       #MyDInt	:= 0;
       #MyWordsinDint[0]	:= "EPICSToPLC"."Word"[#EPICSToPLCDataBlockOffset + 17];
       #MyWordsinDint[1]	:= "EPICSToPLC"."Word"[#EPICSToPLCDataBlockOffset + 18];
       #"P_BlockIcon_LockID" := #MyDInt;    //EPICSName: P_BlockIcon_LockID
    Else
       #DEVICE_PARAM_OK := FALSE; //Invalid Hash
    END_IF;
END_FUNCTION_BLOCK
FUNCTION_BLOCK "DEVTYPE_ICS_HV"
{ S7_Optimized_Access := 'TRUE' }
VERSION : 1.0
   VAR_INPUT
      "OpMode_FreeRun" { ExternalAccessible := 'True'; ExternalVisible := 'False'; ExternalWritable := 'False'; } : BOOL;   //EPICS Status variable: OpMode_FreeRun
      "OpMode_Forced" { ExternalAccessible := 'True'; ExternalVisible := 'False'; ExternalWritable := 'False'; } : BOOL;   //EPICS Status variable: OpMode_Forced
      "Opened" { ExternalAccessible := 'True'; ExternalVisible := 'False'; ExternalWritable := 'False'; } : BOOL;   //EPICS Status variable: Opened
      "Closed" { ExternalAccessible := 'True'; ExternalVisible := 'False'; ExternalWritable := 'False'; } : BOOL;   //EPICS Status variable: Closed
      "ValveColor" { ExternalAccessible := 'True'; ExternalVisible := 'False'; ExternalWritable := 'False'; } : INT;   //EPICS Status variable: ValveColor
      "Inhibit_Manual" { ExternalAccessible := 'True'; ExternalVisible := 'False'; ExternalWritable := 'False'; } : BOOL;   //EPICS Status variable: Inhibit_Manual
      "Inhibit_Force" { ExternalAccessible := 'True'; ExternalVisible := 'False'; ExternalWritable := 'False'; } : BOOL;   //EPICS Status variable: Inhibit_Force
      "Inhibit_Lock" { ExternalAccessible := 'True'; ExternalVisible := 'False'; ExternalWritable := 'False'; } : BOOL;   //EPICS Status variable: Inhibit_Lock
      "EnableFreeRunBtn" { ExternalAccessible := 'True'; ExternalVisible := 'False'; ExternalWritable := 'False'; } : BOOL;   //EPICS Status variable: EnableFreeRunBtn
      "EnableManualBtn" { ExternalAccessible := 'True'; ExternalVisible := 'False'; ExternalWritable := 'False'; } : BOOL;   //EPICS Status variable: EnableManualBtn
      "EnableForcedBtn" { ExternalAccessible := 'True'; ExternalVisible := 'False'; ExternalWritable := 'False'; } : BOOL;   //EPICS Status variable: EnableForcedBtn
      "DevLocked" { ExternalAccessible := 'True'; ExternalVisible := 'False'; ExternalWritable := 'False'; } : BOOL;   //EPICS Status variable: DevLocked
      "Faceplate_LockID" { ExternalAccessible := 'True'; ExternalVisible := 'False'; ExternalWritable := 'False'; } : DINT;   //EPICS Status variable: Faceplate_LockID
      "BlockIcon_LockID" { ExternalAccessible := 'True'; ExternalVisible := 'False'; ExternalWritable := 'False'; } : DINT;   //EPICS Status variable: BlockIcon_LockID
      "LatchAlarm" { ExternalAccessible := 'True'; ExternalVisible := 'False'; ExternalWritable := 'False'; } : BOOL;   //EPICS Status variable: LatchAlarm
      "GroupAlarm" { ExternalAccessible := 'True'; ExternalVisible := 'False'; ExternalWritable := 'False'; } : BOOL;   //EPICS Status variable: GroupAlarm
      "IO_Error" { ExternalAccessible := 'True'; ExternalVisible := 'False'; ExternalWritable := 'False'; } : BOOL;   //EPICS Status variable: IO_Error
      "Input_Module_Error" { ExternalAccessible := 'True'; ExternalVisible := 'False'; ExternalWritable := 'False'; } : BOOL;   //EPICS Status variable: Input_Module_Error
   EPICSToPLCLength { ExternalAccessible := 'False'; ExternalVisible := 'False'; ExternalWritable := 'False'; } : Int;   // Length of device command register array (in words)
   EPICSToPLCDataBlockOffset { ExternalAccessible := 'False'; ExternalVisible := 'False'; ExternalWritable := 'False'; } : Int;   // Offset in EPICS->PLC comms block where this device data resides (in words)
   PLCToEPICSLength { ExternalAccessible := 'False'; ExternalVisible := 'False'; ExternalWritable := 'False'; } : Int;   // Length of device status register array (in words)
   PLCToEPICSDataBlockOffset { ExternalAccessible := 'False'; ExternalVisible := 'False'; ExternalWritable := 'False'; } : Int;   // Offset in PLC->EPICS comms block where this device data resides (in words)
   END_VAR
   VAR_OUTPUT
      "Cmd_FreeRun" { ExternalAccessible := 'True'; ExternalVisible := 'False'; ExternalWritable := 'False'; } : BOOL;   //EPICS Command variable: Cmd_FreeRun
      "Cmd_Force" { ExternalAccessible := 'True'; ExternalVisible := 'False'; ExternalWritable := 'False'; } : BOOL;   //EPICS Command variable: Cmd_Force
      "Cmd_ForceVal" { ExternalAccessible := 'True'; ExternalVisible := 'False'; ExternalWritable := 'False'; } : BOOL;   //EPICS Command variable: Cmd_ForceVal
      "Cmd_AckAlarm" { ExternalAccessible := 'True'; ExternalVisible := 'False'; ExternalWritable := 'False'; } : BOOL;   //EPICS Command variable: Cmd_AckAlarm
      "Cmd_ForceUnlock" { ExternalAccessible := 'True'; ExternalVisible := 'False'; ExternalWritable := 'False'; } : BOOL;   //EPICS Command variable: Cmd_ForceUnlock
      "Cmd_DevLock" { ExternalAccessible := 'True'; ExternalVisible := 'False'; ExternalWritable := 'False'; } : BOOL;   //EPICS Command variable: Cmd_DevLock
      "Cmd_DevUnlock" { ExternalAccessible := 'True'; ExternalVisible := 'False'; ExternalWritable := 'False'; } : BOOL;   //EPICS Command variable: Cmd_DevUnlock
      "P_Faceplate_LockID" { ExternalAccessible := 'True'; ExternalVisible := 'False'; ExternalWritable := 'False'; } : DINT;   //EPICS Parameter variable: P_Faceplate_LockID
      "P_BlockIcon_LockID" { ExternalAccessible := 'True'; ExternalVisible := 'False'; ExternalWritable := 'False'; } : DINT;   //EPICS Parameter variable: P_BlockIcon_LockID
      DEVICE_PARAM_OK { ExternalAccessible := 'False'; ExternalVisible := 'False'; ExternalWritable := 'False'; } : Bool;
   END_VAR
   VAR_IN_OUT
   END_VAR
   Var DB_SPECIFIC
      MyWord { ExternalAccessible := 'False'; ExternalVisible := 'False'; ExternalWritable := 'False'; } : Word;
      MyBytesinWord { ExternalAccessible := 'False'; ExternalVisible := 'False'; ExternalWritable := 'False'; } AT MyWord : Array[0..1] of Byte;
      MyBoolsinWord { ExternalAccessible := 'False'; ExternalVisible := 'False'; ExternalWritable := 'False'; } AT MyWord : Array[0..15] of Bool;
      MyDInt { ExternalAccessible := 'False'; ExternalVisible := 'False'; ExternalWritable := 'False'; } : DInt;
      MyWordsinDint { ExternalAccessible := 'False'; ExternalVisible := 'False'; ExternalWritable := 'False'; } AT MyDInt : Array[0..1] of Word;
      MyReal { ExternalAccessible := 'False'; ExternalVisible := 'False'; ExternalWritable := 'False'; } : Real;
      MyWordsinReal { ExternalAccessible := 'False'; ExternalVisible := 'False'; ExternalWritable := 'False'; } AT MyReal : Array[0..1] of Word;
      MyInt { ExternalAccessible := 'False'; ExternalVisible := 'False'; ExternalWritable := 'False'; } : Int;
      MyWordinInt { ExternalAccessible := 'False'; ExternalVisible := 'False'; ExternalWritable := 'False'; } AT MyInt : Word;
      MyDWord { ExternalAccessible := 'False'; ExternalVisible := 'False'; ExternalWritable := 'False'; } : DWord;
      MyWordsinDWord { ExternalAccessible := 'False'; ExternalVisible := 'False'; ExternalWritable := 'False'; } AT MyDWord : Array[0..1] of Word;
      MyTime { ExternalAccessible := 'False'; ExternalVisible := 'False'; ExternalWritable := 'False'; } : Time;
      MyWordsinTime { ExternalAccessible := 'False'; ExternalVisible := 'False'; ExternalWritable := 'False'; } AT MyTime : Array[0..1] of Word;
      MyString { ExternalAccessible := 'False'; ExternalVisible := 'False'; ExternalWritable := 'False'; } : String[40];
      MyWordsinString { ExternalAccessible := 'False'; ExternalVisible := 'False'; ExternalWritable := 'False'; } AT MyString : Array[0..20] of Word;
   END_VAR
   VAR_TEMP
      HashModbus : DInt;
      HashIFA : DInt;
      HashTIAMap : DInt;
      i : Int;
   END_VAR
    //Author: Miklos Boros (miklos.boros@esss.se), Copyrigth 2017-2020 by European Spallation Source, Lund
    //This block was generated by PLCFactory, please don't change it MANUALLY!
    //Input File Name: Spk-000CDL_Cryo-PLC-010-template-IFA-20220922093722.ifa
    //Generated: 20220922093722
    //According to HASH: 457744924
    //Device type: ICS_HV
    //Description: This function does the variable mapping for a device. All device-variable will be linked to an interface variable defined in this block.

    //********************************************
    //****************HASH check******************
    //********************************************


    #MyWordsinDint[0] := "EPICSToPLC"."Word"[0];
    #MyWordsinDint[1] := "EPICSToPLC"."Word"[1];
    #HashModbus := #MyDInt; //Hash from EPICS/ModbusTCP

    #HashIFA := 457744924; //Hash from Interface Factory as a constant

    #MyWordsinDint[0] := "PLCToEPICS"."Word"[0];
    #MyWordsinDint[1] := "PLCToEPICS"."Word"[1];
    #HashTIAMap := #MyDInt; //Hash from PLCFactory TIA Map


    IF ((#HashIFA = #HashModbus) AND (#HashModbus = #HashTIAMap)) THEN //Check CRCs
        #DEVICE_PARAM_OK := TRUE;
       //##################################### ICS HWI ###############################################
       //############################  ICS Instrument Library     ####################################
       //#  PLC Sample Code in VersionDog: ICS_LIBRARY_MASTER_PLC                                   ##
       //#  CCDB device types: ICS_xxxxx                                                            ##
       //#  EPICS HMI (Block Icons/Faceplates)@ GitLab. Projekt: Cryo / CryogenicsLibrary / CryoLib ##
       //#                                                                                          ##
       //#                          HV - Hand valve with position feedback
       //#                                                                                          ##
       //#                                                                                          ##
       //###########################         Version: 1.3             ################################
       //Author:  Miklos Boros
       //Date:    27-05-2019
       //Version: v1.3
       //Changes:
       //1. Variable Name Unification
       //###########################         Version: 1.0, 1.1, 1.2             ######################
       //Author:  Miklos Boros
       //Date:    28-02-2019
       //Version: v1.2
       //Changes:
       //1. Major review,
       //2. Indent,  unit standardization
       //###########################
       //STATUS BLOCK
       //###########################
       //Operation modes
       //OPI buttons
       //Locking mechanism

    //********************************************
    //*************STATUS VARIABLES***************
    //********************************************


       #MyWord := W#0;
       #MyBoolsinWord[8] := #"OpMode_FreeRun";    //EPICSName: OpMode_FreeRun
       #MyBoolsinWord[9] := #"OpMode_Forced";    //EPICSName: OpMode_Forced
       #MyBoolsinWord[10] := #"Opened";    //EPICSName: Opened
       #MyBoolsinWord[11] := #"Closed";    //EPICSName: Closed
       "PLCToEPICS"."Word"[#PLCToEPICSDataBlockOffset + 0] := #MyWord;

       #MyInt := #"ValveColor";    //EPICSName: ValveColor
       "PLCToEPICS"."Word"[#PLCToEPICSDataBlockOffset + 1] := #MyWordinInt;

       #MyWord := W#0;
       #MyBoolsinWord[8] := #"Inhibit_Manual";    //EPICSName: Inhibit_Manual
       #MyBoolsinWord[9] := #"Inhibit_Force";    //EPICSName: Inhibit_Force
       #MyBoolsinWord[10] := #"Inhibit_Lock";    //EPICSName: Inhibit_Lock
       #MyBoolsinWord[11] := #"EnableFreeRunBtn";    //EPICSName: EnableFreeRunBtn
       #MyBoolsinWord[12] := #"EnableManualBtn";    //EPICSName: EnableManualBtn
       #MyBoolsinWord[13] := #"EnableForcedBtn";    //EPICSName: EnableForcedBtn
       #MyBoolsinWord[14] := #"DevLocked";    //EPICSName: DevLocked
       "PLCToEPICS"."Word"[#PLCToEPICSDataBlockOffset + 2] := #MyWord;

       #MyDInt := #"Faceplate_LockID";    //EPICSName: Faceplate_LockID
       "PLCToEPICS"."Word"[#PLCToEPICSDataBlockOffset + 3] := #MyWordsinDint[0];
       "PLCToEPICS"."Word"[#PLCToEPICSDataBlockOffset + 4] := #MyWordsinDint[1];

       #MyDInt := #"BlockIcon_LockID";    //EPICSName: BlockIcon_LockID
       "PLCToEPICS"."Word"[#PLCToEPICSDataBlockOffset + 5] := #MyWordsinDint[0];
       "PLCToEPICS"."Word"[#PLCToEPICSDataBlockOffset + 6] := #MyWordsinDint[1];

       #MyWord := W#0;
       #MyBoolsinWord[8] := #"LatchAlarm";    //EPICSName: LatchAlarm
       #MyBoolsinWord[9] := #"GroupAlarm";    //EPICSName: GroupAlarm
       #MyBoolsinWord[10] := #"IO_Error";    //EPICSName: IO_Error
       #MyBoolsinWord[11] := #"Input_Module_Error";    //EPICSName: Input_Module_Error
       "PLCToEPICS"."Word"[#PLCToEPICSDataBlockOffset + 7] := #MyWord;

    //********************************************
    //*************COMMAND VARIABLES**************
    //********************************************


       #MyWord := "EPICSToPLC"."Word"[#EPICSToPLCDataBlockOffset + 0];
       "EPICSToPLC"."Word"[#EPICSToPLCDataBlockOffset + 0] := 0;
       #"Cmd_FreeRun" := #MyBoolsinWord[8];    //EPICSName: Cmd_FreeRun
       #"Cmd_Force" := #MyBoolsinWord[9];    //EPICSName: Cmd_Force
       #"Cmd_ForceVal" := #MyBoolsinWord[10];    //EPICSName: Cmd_ForceVal
       #"Cmd_AckAlarm" := #MyBoolsinWord[11];    //EPICSName: Cmd_AckAlarm
       #"Cmd_ForceUnlock" := #MyBoolsinWord[12];    //EPICSName: Cmd_ForceUnlock
       #"Cmd_DevLock" := #MyBoolsinWord[13];    //EPICSName: Cmd_DevLock
       #"Cmd_DevUnlock" := #MyBoolsinWord[14];    //EPICSName: Cmd_DevUnlock

    //********************************************
    //************PARAMETER VARIABLES*************
    //********************************************


       #MyDInt	:= 0;
       #MyWordsinDint[0]	:= "EPICSToPLC"."Word"[#EPICSToPLCDataBlockOffset + 1];
       #MyWordsinDint[1]	:= "EPICSToPLC"."Word"[#EPICSToPLCDataBlockOffset + 2];
       #"P_Faceplate_LockID" := #MyDInt;    //EPICSName: P_Faceplate_LockID

       #MyDInt	:= 0;
       #MyWordsinDint[0]	:= "EPICSToPLC"."Word"[#EPICSToPLCDataBlockOffset + 3];
       #MyWordsinDint[1]	:= "EPICSToPLC"."Word"[#EPICSToPLCDataBlockOffset + 4];
       #"P_BlockIcon_LockID" := #MyDInt;    //EPICSName: P_BlockIcon_LockID
    Else
       #DEVICE_PARAM_OK := FALSE; //Invalid Hash
    END_IF;
END_FUNCTION_BLOCK
FUNCTION_BLOCK "DEVTYPE_ICS_LAKESHORE_TT"
{ S7_Optimized_Access := 'TRUE' }
VERSION : 1.0
   VAR_INPUT
      "OpMode_FreeRun" { ExternalAccessible := 'True'; ExternalVisible := 'False'; ExternalWritable := 'False'; } : BOOL;   //EPICS Status variable: OpMode_FreeRun
      "OpMode_Forced" { ExternalAccessible := 'True'; ExternalVisible := 'False'; ExternalWritable := 'False'; } : BOOL;   //EPICS Status variable: OpMode_Forced
      "Inhibit_Manual" { ExternalAccessible := 'True'; ExternalVisible := 'False'; ExternalWritable := 'False'; } : BOOL;   //EPICS Status variable: Inhibit_Manual
      "Inhibit_Force" { ExternalAccessible := 'True'; ExternalVisible := 'False'; ExternalWritable := 'False'; } : BOOL;   //EPICS Status variable: Inhibit_Force
      "Inhibit_Lock" { ExternalAccessible := 'True'; ExternalVisible := 'False'; ExternalWritable := 'False'; } : BOOL;   //EPICS Status variable: Inhibit_Lock
      "TransmitterColor" { ExternalAccessible := 'True'; ExternalVisible := 'False'; ExternalWritable := 'False'; } : INT;   //EPICS Status variable: TransmitterColor
      "MinTemp" { ExternalAccessible := 'True'; ExternalVisible := 'False'; ExternalWritable := 'False'; } : REAL;   //EPICS Status variable: MinTemp
      "MaxTemp" { ExternalAccessible := 'True'; ExternalVisible := 'False'; ExternalWritable := 'False'; } : REAL;   //EPICS Status variable: MaxTemp
      "EnableFreeRunBtn" { ExternalAccessible := 'True'; ExternalVisible := 'False'; ExternalWritable := 'False'; } : BOOL;   //EPICS Status variable: EnableFreeRunBtn
      "EnableForcedBtn" { ExternalAccessible := 'True'; ExternalVisible := 'False'; ExternalWritable := 'False'; } : BOOL;   //EPICS Status variable: EnableForcedBtn
      "EnableManualBtn" { ExternalAccessible := 'True'; ExternalVisible := 'False'; ExternalWritable := 'False'; } : BOOL;   //EPICS Status variable: EnableManualBtn
      "MeasValue" { ExternalAccessible := 'True'; ExternalVisible := 'False'; ExternalWritable := 'False'; } : REAL;   //EPICS Status variable: MeasValue
      "DevLocked" { ExternalAccessible := 'True'; ExternalVisible := 'False'; ExternalWritable := 'False'; } : BOOL;   //EPICS Status variable: DevLocked
      "Faceplate_LockID" { ExternalAccessible := 'True'; ExternalVisible := 'False'; ExternalWritable := 'False'; } : DINT;   //EPICS Status variable: Faceplate_LockID
      "BlockIcon_LockID" { ExternalAccessible := 'True'; ExternalVisible := 'False'; ExternalWritable := 'False'; } : DINT;   //EPICS Status variable: BlockIcon_LockID
      "LatchAlarm" { ExternalAccessible := 'True'; ExternalVisible := 'False'; ExternalWritable := 'False'; } : BOOL;   //EPICS Status variable: LatchAlarm
      "GroupAlarm" { ExternalAccessible := 'True'; ExternalVisible := 'False'; ExternalWritable := 'False'; } : BOOL;   //EPICS Status variable: GroupAlarm
      "Underrange" { ExternalAccessible := 'True'; ExternalVisible := 'False'; ExternalWritable := 'False'; } : BOOL;   //EPICS Status variable: Underrange
      "Overrange" { ExternalAccessible := 'True'; ExternalVisible := 'False'; ExternalWritable := 'False'; } : BOOL;   //EPICS Status variable: Overrange
      "HIHI" { ExternalAccessible := 'True'; ExternalVisible := 'False'; ExternalWritable := 'False'; } : BOOL;   //EPICS Status variable: HIHI
      "HI" { ExternalAccessible := 'True'; ExternalVisible := 'False'; ExternalWritable := 'False'; } : BOOL;   //EPICS Status variable: HI
      "LO" { ExternalAccessible := 'True'; ExternalVisible := 'False'; ExternalWritable := 'False'; } : BOOL;   //EPICS Status variable: LO
      "LOLO" { ExternalAccessible := 'True'; ExternalVisible := 'False'; ExternalWritable := 'False'; } : BOOL;   //EPICS Status variable: LOLO
      "Param_Error" { ExternalAccessible := 'True'; ExternalVisible := 'False'; ExternalWritable := 'False'; } : BOOL;   //EPICS Status variable: Param_Error
      "PN_Module_Error" { ExternalAccessible := 'True'; ExternalVisible := 'False'; ExternalWritable := 'False'; } : BOOL;   //EPICS Status variable: PN_Module_Error
      "FB_ForceValue" { ExternalAccessible := 'True'; ExternalVisible := 'False'; ExternalWritable := 'False'; } : REAL;   //EPICS Status variable: FB_ForceValue
      "FB_Limit_HIHI" { ExternalAccessible := 'True'; ExternalVisible := 'False'; ExternalWritable := 'False'; } : REAL;   //EPICS Status variable: FB_Limit_HIHI
      "FB_Limit_HI" { ExternalAccessible := 'True'; ExternalVisible := 'False'; ExternalWritable := 'False'; } : REAL;   //EPICS Status variable: FB_Limit_HI
      "FB_Limit_LO" { ExternalAccessible := 'True'; ExternalVisible := 'False'; ExternalWritable := 'False'; } : REAL;   //EPICS Status variable: FB_Limit_LO
      "FB_Limit_LOLO" { ExternalAccessible := 'True'; ExternalVisible := 'False'; ExternalWritable := 'False'; } : REAL;   //EPICS Status variable: FB_Limit_LOLO
   EPICSToPLCLength { ExternalAccessible := 'False'; ExternalVisible := 'False'; ExternalWritable := 'False'; } : Int;   // Length of device command register array (in words)
   EPICSToPLCDataBlockOffset { ExternalAccessible := 'False'; ExternalVisible := 'False'; ExternalWritable := 'False'; } : Int;   // Offset in EPICS->PLC comms block where this device data resides (in words)
   PLCToEPICSLength { ExternalAccessible := 'False'; ExternalVisible := 'False'; ExternalWritable := 'False'; } : Int;   // Length of device status register array (in words)
   PLCToEPICSDataBlockOffset { ExternalAccessible := 'False'; ExternalVisible := 'False'; ExternalWritable := 'False'; } : Int;   // Offset in PLC->EPICS comms block where this device data resides (in words)
   END_VAR
   VAR_OUTPUT
      "Cmd_FreeRun" { ExternalAccessible := 'True'; ExternalVisible := 'False'; ExternalWritable := 'False'; } : BOOL;   //EPICS Command variable: Cmd_FreeRun
      "Cmd_Force" { ExternalAccessible := 'True'; ExternalVisible := 'False'; ExternalWritable := 'False'; } : BOOL;   //EPICS Command variable: Cmd_Force
      "Cmd_ForceVal" { ExternalAccessible := 'True'; ExternalVisible := 'False'; ExternalWritable := 'False'; } : BOOL;   //EPICS Command variable: Cmd_ForceVal
      "Cmd_AckAlarm" { ExternalAccessible := 'True'; ExternalVisible := 'False'; ExternalWritable := 'False'; } : BOOL;   //EPICS Command variable: Cmd_AckAlarm
      "Cmd_ForceUnlock" { ExternalAccessible := 'True'; ExternalVisible := 'False'; ExternalWritable := 'False'; } : BOOL;   //EPICS Command variable: Cmd_ForceUnlock
      "Cmd_DevLock" { ExternalAccessible := 'True'; ExternalVisible := 'False'; ExternalWritable := 'False'; } : BOOL;   //EPICS Command variable: Cmd_DevLock
      "Cmd_DevUnlock" { ExternalAccessible := 'True'; ExternalVisible := 'False'; ExternalWritable := 'False'; } : BOOL;   //EPICS Command variable: Cmd_DevUnlock
      "P_Limit_HIHI" { ExternalAccessible := 'True'; ExternalVisible := 'False'; ExternalWritable := 'False'; } : REAL;   //EPICS Parameter variable: P_Limit_HIHI
      "P_Limit_HI" { ExternalAccessible := 'True'; ExternalVisible := 'False'; ExternalWritable := 'False'; } : REAL;   //EPICS Parameter variable: P_Limit_HI
      "P_Limit_LO" { ExternalAccessible := 'True'; ExternalVisible := 'False'; ExternalWritable := 'False'; } : REAL;   //EPICS Parameter variable: P_Limit_LO
      "P_Limit_LOLO" { ExternalAccessible := 'True'; ExternalVisible := 'False'; ExternalWritable := 'False'; } : REAL;   //EPICS Parameter variable: P_Limit_LOLO
      "P_ForceValue" { ExternalAccessible := 'True'; ExternalVisible := 'False'; ExternalWritable := 'False'; } : REAL;   //EPICS Parameter variable: P_ForceValue
      "P_Faceplate_LockID" { ExternalAccessible := 'True'; ExternalVisible := 'False'; ExternalWritable := 'False'; } : DINT;   //EPICS Parameter variable: P_Faceplate_LockID
      "P_BlockIcon_LockID" { ExternalAccessible := 'True'; ExternalVisible := 'False'; ExternalWritable := 'False'; } : DINT;   //EPICS Parameter variable: P_BlockIcon_LockID
      DEVICE_PARAM_OK { ExternalAccessible := 'False'; ExternalVisible := 'False'; ExternalWritable := 'False'; } : Bool;
   END_VAR
   VAR_IN_OUT
   END_VAR
   Var DB_SPECIFIC
      MyWord { ExternalAccessible := 'False'; ExternalVisible := 'False'; ExternalWritable := 'False'; } : Word;
      MyBytesinWord { ExternalAccessible := 'False'; ExternalVisible := 'False'; ExternalWritable := 'False'; } AT MyWord : Array[0..1] of Byte;
      MyBoolsinWord { ExternalAccessible := 'False'; ExternalVisible := 'False'; ExternalWritable := 'False'; } AT MyWord : Array[0..15] of Bool;
      MyDInt { ExternalAccessible := 'False'; ExternalVisible := 'False'; ExternalWritable := 'False'; } : DInt;
      MyWordsinDint { ExternalAccessible := 'False'; ExternalVisible := 'False'; ExternalWritable := 'False'; } AT MyDInt : Array[0..1] of Word;
      MyReal { ExternalAccessible := 'False'; ExternalVisible := 'False'; ExternalWritable := 'False'; } : Real;
      MyWordsinReal { ExternalAccessible := 'False'; ExternalVisible := 'False'; ExternalWritable := 'False'; } AT MyReal : Array[0..1] of Word;
      MyInt { ExternalAccessible := 'False'; ExternalVisible := 'False'; ExternalWritable := 'False'; } : Int;
      MyWordinInt { ExternalAccessible := 'False'; ExternalVisible := 'False'; ExternalWritable := 'False'; } AT MyInt : Word;
      MyDWord { ExternalAccessible := 'False'; ExternalVisible := 'False'; ExternalWritable := 'False'; } : DWord;
      MyWordsinDWord { ExternalAccessible := 'False'; ExternalVisible := 'False'; ExternalWritable := 'False'; } AT MyDWord : Array[0..1] of Word;
      MyTime { ExternalAccessible := 'False'; ExternalVisible := 'False'; ExternalWritable := 'False'; } : Time;
      MyWordsinTime { ExternalAccessible := 'False'; ExternalVisible := 'False'; ExternalWritable := 'False'; } AT MyTime : Array[0..1] of Word;
      MyString { ExternalAccessible := 'False'; ExternalVisible := 'False'; ExternalWritable := 'False'; } : String[40];
      MyWordsinString { ExternalAccessible := 'False'; ExternalVisible := 'False'; ExternalWritable := 'False'; } AT MyString : Array[0..20] of Word;
   END_VAR
   VAR_TEMP
      HashModbus : DInt;
      HashIFA : DInt;
      HashTIAMap : DInt;
      i : Int;
   END_VAR
    //Author: Miklos Boros (miklos.boros@esss.se), Copyrigth 2017-2020 by European Spallation Source, Lund
    //This block was generated by PLCFactory, please don't change it MANUALLY!
    //Input File Name: Spk-000CDL_Cryo-PLC-010-template-IFA-20220922093722.ifa
    //Generated: 20220922093722
    //According to HASH: 457744924
    //Device type: ICS_LAKESHORE_TT
    //Description: This function does the variable mapping for a device. All device-variable will be linked to an interface variable defined in this block.

    //********************************************
    //****************HASH check******************
    //********************************************


    #MyWordsinDint[0] := "EPICSToPLC"."Word"[0];
    #MyWordsinDint[1] := "EPICSToPLC"."Word"[1];
    #HashModbus := #MyDInt; //Hash from EPICS/ModbusTCP

    #HashIFA := 457744924; //Hash from Interface Factory as a constant

    #MyWordsinDint[0] := "PLCToEPICS"."Word"[0];
    #MyWordsinDint[1] := "PLCToEPICS"."Word"[1];
    #HashTIAMap := #MyDInt; //Hash from PLCFactory TIA Map


    IF ((#HashIFA = #HashModbus) AND (#HashModbus = #HashTIAMap)) THEN //Check CRCs
        #DEVICE_PARAM_OK := TRUE;
       //##################################### ICS HWI ###############################################
       //############################  ICS Instrument Library     ####################################
       //#  PLC Sample Code in VersionDog: ICS_LIBRARY_MASTER_PLC                                   ##
       //#  CCDB device types: ICS_xxxxx                                                            ##
       //#  EPICS HMI (Block Icons/Faceplates)@ GitLab. Projekt: Cryo / CryogenicsLibrary / CryoLib ##
       //#                                                                                          ##
       //#                      TT - Temperature Transmitter in K with Lakeshore                    ##
       //#                                                                                          ##
       //#                                                                                          ##
       //###########################         Version: 1.4             ################################
       //Author:  Miklos Boros
       //Date:    16-12-2019
       //Version: v1.4
       //Changes:
       //1. Modified TT for direct Temp measurement with Lakeshore
       //###########################         Version: 1.3             ################################
       //Author:  Miklos Boros
       //Date:    27-05-2019
       //Version: v1.3
       //Changes:
       //1. Variable Name Unification
       //###########################         Version: 1.2             ################################
       //Author:  Miklos Boros
       //Date:    28-02-2019
       //Version: v1.2
       //Changes:
       //1. Major review,
       //2. Indent,  unit standardization
       //###########################         Version: 1.1             ################################
       //Author:  Miklos Boros, Marino Vojneski
       //Date:    12-06-2018
       //Version: v1.1
       //Changes:
       //1. Modified Alarm Signal section to be compatible with new format.
       //########################### Version: 1.0             ########################################
       //Author:  Miklos Boros
       //Date:    25-01-2018
       //Version: v1.0
       //###########################
       //STATUS BLOCK
       //###########################
       //Operation modes
       //OPI buttons
       //Limits

    //********************************************
    //*************STATUS VARIABLES***************
    //********************************************


       #MyWord := W#0;
       #MyBoolsinWord[8] := #"OpMode_FreeRun";    //EPICSName: OpMode_FreeRun
       #MyBoolsinWord[9] := #"OpMode_Forced";    //EPICSName: OpMode_Forced
       #MyBoolsinWord[10] := #"Inhibit_Manual";    //EPICSName: Inhibit_Manual
       #MyBoolsinWord[11] := #"Inhibit_Force";    //EPICSName: Inhibit_Force
       #MyBoolsinWord[12] := #"Inhibit_Lock";    //EPICSName: Inhibit_Lock
       "PLCToEPICS"."Word"[#PLCToEPICSDataBlockOffset + 0] := #MyWord;

       #MyInt := #"TransmitterColor";    //EPICSName: TransmitterColor
       "PLCToEPICS"."Word"[#PLCToEPICSDataBlockOffset + 1] := #MyWordinInt;

       #MyReal := #"MinTemp";    //EPICSName: MinTemp
       "PLCToEPICS"."Word"[#PLCToEPICSDataBlockOffset + 2] := #MyWordsinReal[0];
       "PLCToEPICS"."Word"[#PLCToEPICSDataBlockOffset + 3] := #MyWordsinReal[1];

       #MyReal := #"MaxTemp";    //EPICSName: MaxTemp
       "PLCToEPICS"."Word"[#PLCToEPICSDataBlockOffset + 4] := #MyWordsinReal[0];
       "PLCToEPICS"."Word"[#PLCToEPICSDataBlockOffset + 5] := #MyWordsinReal[1];

       #MyWord := W#0;
       #MyBoolsinWord[8] := #"EnableFreeRunBtn";    //EPICSName: EnableFreeRunBtn
       #MyBoolsinWord[9] := #"EnableForcedBtn";    //EPICSName: EnableForcedBtn
       #MyBoolsinWord[10] := #"EnableManualBtn";    //EPICSName: EnableManualBtn
       "PLCToEPICS"."Word"[#PLCToEPICSDataBlockOffset + 6] := #MyWord;

       #MyReal := #"MeasValue";    //EPICSName: MeasValue
       "PLCToEPICS"."Word"[#PLCToEPICSDataBlockOffset + 7] := #MyWordsinReal[0];
       "PLCToEPICS"."Word"[#PLCToEPICSDataBlockOffset + 8] := #MyWordsinReal[1];

       #MyWord := W#0;
       #MyBoolsinWord[8] := #"DevLocked";    //EPICSName: DevLocked
       "PLCToEPICS"."Word"[#PLCToEPICSDataBlockOffset + 9] := #MyWord;

       #MyDInt := #"Faceplate_LockID";    //EPICSName: Faceplate_LockID
       "PLCToEPICS"."Word"[#PLCToEPICSDataBlockOffset + 10] := #MyWordsinDint[0];
       "PLCToEPICS"."Word"[#PLCToEPICSDataBlockOffset + 11] := #MyWordsinDint[1];

       #MyDInt := #"BlockIcon_LockID";    //EPICSName: BlockIcon_LockID
       "PLCToEPICS"."Word"[#PLCToEPICSDataBlockOffset + 12] := #MyWordsinDint[0];
       "PLCToEPICS"."Word"[#PLCToEPICSDataBlockOffset + 13] := #MyWordsinDint[1];

       #MyWord := W#0;
       #MyBoolsinWord[8] := #"LatchAlarm";    //EPICSName: LatchAlarm
       #MyBoolsinWord[9] := #"GroupAlarm";    //EPICSName: GroupAlarm
       #MyBoolsinWord[10] := #"Underrange";    //EPICSName: Underrange
       #MyBoolsinWord[11] := #"Overrange";    //EPICSName: Overrange
       #MyBoolsinWord[12] := #"HIHI";    //EPICSName: HIHI
       #MyBoolsinWord[13] := #"HI";    //EPICSName: HI
       #MyBoolsinWord[14] := #"LO";    //EPICSName: LO
       #MyBoolsinWord[15] := #"LOLO";    //EPICSName: LOLO
       #MyBoolsinWord[0] := #"Param_Error";    //EPICSName: Param_Error
       #MyBoolsinWord[1] := #"PN_Module_Error";    //EPICSName: PN_Module_Error
       "PLCToEPICS"."Word"[#PLCToEPICSDataBlockOffset + 14] := #MyWord;

       #MyReal := #"FB_ForceValue";    //EPICSName: FB_ForceValue
       "PLCToEPICS"."Word"[#PLCToEPICSDataBlockOffset + 15] := #MyWordsinReal[0];
       "PLCToEPICS"."Word"[#PLCToEPICSDataBlockOffset + 16] := #MyWordsinReal[1];

       #MyReal := #"FB_Limit_HIHI";    //EPICSName: FB_Limit_HIHI
       "PLCToEPICS"."Word"[#PLCToEPICSDataBlockOffset + 17] := #MyWordsinReal[0];
       "PLCToEPICS"."Word"[#PLCToEPICSDataBlockOffset + 18] := #MyWordsinReal[1];

       #MyReal := #"FB_Limit_HI";    //EPICSName: FB_Limit_HI
       "PLCToEPICS"."Word"[#PLCToEPICSDataBlockOffset + 19] := #MyWordsinReal[0];
       "PLCToEPICS"."Word"[#PLCToEPICSDataBlockOffset + 20] := #MyWordsinReal[1];

       #MyReal := #"FB_Limit_LO";    //EPICSName: FB_Limit_LO
       "PLCToEPICS"."Word"[#PLCToEPICSDataBlockOffset + 21] := #MyWordsinReal[0];
       "PLCToEPICS"."Word"[#PLCToEPICSDataBlockOffset + 22] := #MyWordsinReal[1];

       #MyReal := #"FB_Limit_LOLO";    //EPICSName: FB_Limit_LOLO
       "PLCToEPICS"."Word"[#PLCToEPICSDataBlockOffset + 23] := #MyWordsinReal[0];
       "PLCToEPICS"."Word"[#PLCToEPICSDataBlockOffset + 24] := #MyWordsinReal[1];

    //********************************************
    //*************COMMAND VARIABLES**************
    //********************************************


       #MyWord := "EPICSToPLC"."Word"[#EPICSToPLCDataBlockOffset + 0];
       "EPICSToPLC"."Word"[#EPICSToPLCDataBlockOffset + 0] := 0;
       #"Cmd_FreeRun" := #MyBoolsinWord[8];    //EPICSName: Cmd_FreeRun
       #"Cmd_Force" := #MyBoolsinWord[9];    //EPICSName: Cmd_Force
       #"Cmd_ForceVal" := #MyBoolsinWord[10];    //EPICSName: Cmd_ForceVal
       #"Cmd_AckAlarm" := #MyBoolsinWord[11];    //EPICSName: Cmd_AckAlarm
       #"Cmd_ForceUnlock" := #MyBoolsinWord[12];    //EPICSName: Cmd_ForceUnlock
       #"Cmd_DevLock" := #MyBoolsinWord[13];    //EPICSName: Cmd_DevLock
       #"Cmd_DevUnlock" := #MyBoolsinWord[14];    //EPICSName: Cmd_DevUnlock

    //********************************************
    //************PARAMETER VARIABLES*************
    //********************************************


       #MyReal	:= 0.0;
       #MyWordsinReal[0]	:= "EPICSToPLC"."Word"[#EPICSToPLCDataBlockOffset + 1];
       #MyWordsinReal[1]	:= "EPICSToPLC"."Word"[#EPICSToPLCDataBlockOffset + 2];
       #"P_Limit_HIHI" := #MyReal;    //EPICSName: P_Limit_HIHI

       #MyReal	:= 0.0;
       #MyWordsinReal[0]	:= "EPICSToPLC"."Word"[#EPICSToPLCDataBlockOffset + 3];
       #MyWordsinReal[1]	:= "EPICSToPLC"."Word"[#EPICSToPLCDataBlockOffset + 4];
       #"P_Limit_HI" := #MyReal;    //EPICSName: P_Limit_HI

       #MyReal	:= 0.0;
       #MyWordsinReal[0]	:= "EPICSToPLC"."Word"[#EPICSToPLCDataBlockOffset + 5];
       #MyWordsinReal[1]	:= "EPICSToPLC"."Word"[#EPICSToPLCDataBlockOffset + 6];
       #"P_Limit_LO" := #MyReal;    //EPICSName: P_Limit_LO

       #MyReal	:= 0.0;
       #MyWordsinReal[0]	:= "EPICSToPLC"."Word"[#EPICSToPLCDataBlockOffset + 7];
       #MyWordsinReal[1]	:= "EPICSToPLC"."Word"[#EPICSToPLCDataBlockOffset + 8];
       #"P_Limit_LOLO" := #MyReal;    //EPICSName: P_Limit_LOLO

       #MyReal	:= 0.0;
       #MyWordsinReal[0]	:= "EPICSToPLC"."Word"[#EPICSToPLCDataBlockOffset + 9];
       #MyWordsinReal[1]	:= "EPICSToPLC"."Word"[#EPICSToPLCDataBlockOffset + 10];
       #"P_ForceValue" := #MyReal;    //EPICSName: P_ForceValue

       #MyDInt	:= 0;
       #MyWordsinDint[0]	:= "EPICSToPLC"."Word"[#EPICSToPLCDataBlockOffset + 11];
       #MyWordsinDint[1]	:= "EPICSToPLC"."Word"[#EPICSToPLCDataBlockOffset + 12];
       #"P_Faceplate_LockID" := #MyDInt;    //EPICSName: P_Faceplate_LockID

       #MyDInt	:= 0;
       #MyWordsinDint[0]	:= "EPICSToPLC"."Word"[#EPICSToPLCDataBlockOffset + 13];
       #MyWordsinDint[1]	:= "EPICSToPLC"."Word"[#EPICSToPLCDataBlockOffset + 14];
       #"P_BlockIcon_LockID" := #MyDInt;    //EPICSName: P_BlockIcon_LockID
    Else
       #DEVICE_PARAM_OK := FALSE; //Invalid Hash
    END_IF;
END_FUNCTION_BLOCK
FUNCTION_BLOCK "DEVTYPE_ICS_LT"
{ S7_Optimized_Access := 'TRUE' }
VERSION : 1.0
   VAR_INPUT
      "OpMode_FreeRun" { ExternalAccessible := 'True'; ExternalVisible := 'False'; ExternalWritable := 'False'; } : BOOL;   //EPICS Status variable: OpMode_FreeRun
      "OpMode_Forced" { ExternalAccessible := 'True'; ExternalVisible := 'False'; ExternalWritable := 'False'; } : BOOL;   //EPICS Status variable: OpMode_Forced
      "Inhibit_Manual" { ExternalAccessible := 'True'; ExternalVisible := 'False'; ExternalWritable := 'False'; } : BOOL;   //EPICS Status variable: Inhibit_Manual
      "Inhibit_Force" { ExternalAccessible := 'True'; ExternalVisible := 'False'; ExternalWritable := 'False'; } : BOOL;   //EPICS Status variable: Inhibit_Force
      "Inhibit_Lock" { ExternalAccessible := 'True'; ExternalVisible := 'False'; ExternalWritable := 'False'; } : BOOL;   //EPICS Status variable: Inhibit_Lock
      "TransmitterColor" { ExternalAccessible := 'True'; ExternalVisible := 'False'; ExternalWritable := 'False'; } : INT;   //EPICS Status variable: TransmitterColor
      "EnableFreeRunBtn" { ExternalAccessible := 'True'; ExternalVisible := 'False'; ExternalWritable := 'False'; } : BOOL;   //EPICS Status variable: EnableFreeRunBtn
      "EnableForcedBtn" { ExternalAccessible := 'True'; ExternalVisible := 'False'; ExternalWritable := 'False'; } : BOOL;   //EPICS Status variable: EnableForcedBtn
      "EnableManualBtn" { ExternalAccessible := 'True'; ExternalVisible := 'False'; ExternalWritable := 'False'; } : BOOL;   //EPICS Status variable: EnableManualBtn
      "ScaleLOW" { ExternalAccessible := 'True'; ExternalVisible := 'False'; ExternalWritable := 'False'; } : REAL;   //EPICS Status variable: ScaleLOW
      "ScaleHIGH" { ExternalAccessible := 'True'; ExternalVisible := 'False'; ExternalWritable := 'False'; } : REAL;   //EPICS Status variable: ScaleHIGH
      "MeasValue" { ExternalAccessible := 'True'; ExternalVisible := 'False'; ExternalWritable := 'False'; } : REAL;   //EPICS Status variable: MeasValue
      "RAWValue" { ExternalAccessible := 'True'; ExternalVisible := 'False'; ExternalWritable := 'False'; } : REAL;   //EPICS Status variable: RAWValue
      "DevLocked" { ExternalAccessible := 'True'; ExternalVisible := 'False'; ExternalWritable := 'False'; } : BOOL;   //EPICS Status variable: DevLocked
      "Faceplate_LockID" { ExternalAccessible := 'True'; ExternalVisible := 'False'; ExternalWritable := 'False'; } : DINT;   //EPICS Status variable: Faceplate_LockID
      "BlockIcon_LockID" { ExternalAccessible := 'True'; ExternalVisible := 'False'; ExternalWritable := 'False'; } : DINT;   //EPICS Status variable: BlockIcon_LockID
      "LatchAlarm" { ExternalAccessible := 'True'; ExternalVisible := 'False'; ExternalWritable := 'False'; } : BOOL;   //EPICS Status variable: LatchAlarm
      "GroupAlarm" { ExternalAccessible := 'True'; ExternalVisible := 'False'; ExternalWritable := 'False'; } : BOOL;   //EPICS Status variable: GroupAlarm
      "Underrange" { ExternalAccessible := 'True'; ExternalVisible := 'False'; ExternalWritable := 'False'; } : BOOL;   //EPICS Status variable: Underrange
      "Overrange" { ExternalAccessible := 'True'; ExternalVisible := 'False'; ExternalWritable := 'False'; } : BOOL;   //EPICS Status variable: Overrange
      "HIHI" { ExternalAccessible := 'True'; ExternalVisible := 'False'; ExternalWritable := 'False'; } : BOOL;   //EPICS Status variable: HIHI
      "HI" { ExternalAccessible := 'True'; ExternalVisible := 'False'; ExternalWritable := 'False'; } : BOOL;   //EPICS Status variable: HI
      "LO" { ExternalAccessible := 'True'; ExternalVisible := 'False'; ExternalWritable := 'False'; } : BOOL;   //EPICS Status variable: LO
      "LOLO" { ExternalAccessible := 'True'; ExternalVisible := 'False'; ExternalWritable := 'False'; } : BOOL;   //EPICS Status variable: LOLO
      "IO_Error" { ExternalAccessible := 'True'; ExternalVisible := 'False'; ExternalWritable := 'False'; } : BOOL;   //EPICS Status variable: IO_Error
      "Module_Error" { ExternalAccessible := 'True'; ExternalVisible := 'False'; ExternalWritable := 'False'; } : BOOL;   //EPICS Status variable: Module_Error
      "Param_Error" { ExternalAccessible := 'True'; ExternalVisible := 'False'; ExternalWritable := 'False'; } : BOOL;   //EPICS Status variable: Param_Error
      "FB_ForceValue" { ExternalAccessible := 'True'; ExternalVisible := 'False'; ExternalWritable := 'False'; } : REAL;   //EPICS Status variable: FB_ForceValue
      "FB_Limit_HIHI" { ExternalAccessible := 'True'; ExternalVisible := 'False'; ExternalWritable := 'False'; } : REAL;   //EPICS Status variable: FB_Limit_HIHI
      "FB_Limit_HI" { ExternalAccessible := 'True'; ExternalVisible := 'False'; ExternalWritable := 'False'; } : REAL;   //EPICS Status variable: FB_Limit_HI
      "FB_Limit_LO" { ExternalAccessible := 'True'; ExternalVisible := 'False'; ExternalWritable := 'False'; } : REAL;   //EPICS Status variable: FB_Limit_LO
      "FB_Limit_LOLO" { ExternalAccessible := 'True'; ExternalVisible := 'False'; ExternalWritable := 'False'; } : REAL;   //EPICS Status variable: FB_Limit_LOLO
      "Timer_enabled" { ExternalAccessible := 'True'; ExternalVisible := 'False'; ExternalWritable := 'False'; } : BOOL;   //EPICS Status variable: Timer_enabled
      "T_triggered" { ExternalAccessible := 'True'; ExternalVisible := 'False'; ExternalWritable := 'False'; } : BOOL;   //EPICS Status variable: T_triggered
      "T_running" { ExternalAccessible := 'True'; ExternalVisible := 'False'; ExternalWritable := 'False'; } : INT;   //EPICS Status variable: T_running
      "F_enabled" { ExternalAccessible := 'True'; ExternalVisible := 'False'; ExternalWritable := 'False'; } : BOOL;   //EPICS Status variable: F_enabled
      "FiltedValue" { ExternalAccessible := 'True'; ExternalVisible := 'False'; ExternalWritable := 'False'; } : REAL;   //EPICS Status variable: FiltedValue
   EPICSToPLCLength { ExternalAccessible := 'False'; ExternalVisible := 'False'; ExternalWritable := 'False'; } : Int;   // Length of device command register array (in words)
   EPICSToPLCDataBlockOffset { ExternalAccessible := 'False'; ExternalVisible := 'False'; ExternalWritable := 'False'; } : Int;   // Offset in EPICS->PLC comms block where this device data resides (in words)
   PLCToEPICSLength { ExternalAccessible := 'False'; ExternalVisible := 'False'; ExternalWritable := 'False'; } : Int;   // Length of device status register array (in words)
   PLCToEPICSDataBlockOffset { ExternalAccessible := 'False'; ExternalVisible := 'False'; ExternalWritable := 'False'; } : Int;   // Offset in PLC->EPICS comms block where this device data resides (in words)
   END_VAR
   VAR_OUTPUT
      "Cmd_FreeRun" { ExternalAccessible := 'True'; ExternalVisible := 'False'; ExternalWritable := 'False'; } : BOOL;   //EPICS Command variable: Cmd_FreeRun
      "Cmd_Force" { ExternalAccessible := 'True'; ExternalVisible := 'False'; ExternalWritable := 'False'; } : BOOL;   //EPICS Command variable: Cmd_Force
      "Cmd_ForceVal" { ExternalAccessible := 'True'; ExternalVisible := 'False'; ExternalWritable := 'False'; } : BOOL;   //EPICS Command variable: Cmd_ForceVal
      "Cmd_AckAlarm" { ExternalAccessible := 'True'; ExternalVisible := 'False'; ExternalWritable := 'False'; } : BOOL;   //EPICS Command variable: Cmd_AckAlarm
      "Cmd_ForceUnlock" { ExternalAccessible := 'True'; ExternalVisible := 'False'; ExternalWritable := 'False'; } : BOOL;   //EPICS Command variable: Cmd_ForceUnlock
      "Cmd_DevLock" { ExternalAccessible := 'True'; ExternalVisible := 'False'; ExternalWritable := 'False'; } : BOOL;   //EPICS Command variable: Cmd_DevLock
      "Cmd_DevUnlock" { ExternalAccessible := 'True'; ExternalVisible := 'False'; ExternalWritable := 'False'; } : BOOL;   //EPICS Command variable: Cmd_DevUnlock
      "P_Limit_HIHI" { ExternalAccessible := 'True'; ExternalVisible := 'False'; ExternalWritable := 'False'; } : REAL;   //EPICS Parameter variable: P_Limit_HIHI
      "P_Limit_HI" { ExternalAccessible := 'True'; ExternalVisible := 'False'; ExternalWritable := 'False'; } : REAL;   //EPICS Parameter variable: P_Limit_HI
      "P_Limit_LO" { ExternalAccessible := 'True'; ExternalVisible := 'False'; ExternalWritable := 'False'; } : REAL;   //EPICS Parameter variable: P_Limit_LO
      "P_Limit_LOLO" { ExternalAccessible := 'True'; ExternalVisible := 'False'; ExternalWritable := 'False'; } : REAL;   //EPICS Parameter variable: P_Limit_LOLO
      "P_ForceValue" { ExternalAccessible := 'True'; ExternalVisible := 'False'; ExternalWritable := 'False'; } : REAL;   //EPICS Parameter variable: P_ForceValue
      "P_Faceplate_LockID" { ExternalAccessible := 'True'; ExternalVisible := 'False'; ExternalWritable := 'False'; } : DINT;   //EPICS Parameter variable: P_Faceplate_LockID
      "P_BlockIcon_LockID" { ExternalAccessible := 'True'; ExternalVisible := 'False'; ExternalWritable := 'False'; } : DINT;   //EPICS Parameter variable: P_BlockIcon_LockID
      "T_period" { ExternalAccessible := 'True'; ExternalVisible := 'False'; ExternalWritable := 'False'; } : INT;   //EPICS Parameter variable: T_period
      "F_interval" { ExternalAccessible := 'True'; ExternalVisible := 'False'; ExternalWritable := 'False'; } : INT;   //EPICS Parameter variable: F_interval
      "F_buffer" { ExternalAccessible := 'True'; ExternalVisible := 'False'; ExternalWritable := 'False'; } : INT;   //EPICS Parameter variable: F_buffer
      "F_Enable" { ExternalAccessible := 'True'; ExternalVisible := 'False'; ExternalWritable := 'False'; } : BOOL;   //EPICS Parameter variable: F_Enable
      "P_RampUPSpeed" { ExternalAccessible := 'True'; ExternalVisible := 'False'; ExternalWritable := 'False'; } : REAL;   //EPICS Parameter variable: P_RampUPSpeed
      "P_RampDNSpeed" { ExternalAccessible := 'True'; ExternalVisible := 'False'; ExternalWritable := 'False'; } : REAL;   //EPICS Parameter variable: P_RampDNSpeed
      DEVICE_PARAM_OK { ExternalAccessible := 'False'; ExternalVisible := 'False'; ExternalWritable := 'False'; } : Bool;
   END_VAR
   VAR_IN_OUT
   END_VAR
   Var DB_SPECIFIC
      MyWord { ExternalAccessible := 'False'; ExternalVisible := 'False'; ExternalWritable := 'False'; } : Word;
      MyBytesinWord { ExternalAccessible := 'False'; ExternalVisible := 'False'; ExternalWritable := 'False'; } AT MyWord : Array[0..1] of Byte;
      MyBoolsinWord { ExternalAccessible := 'False'; ExternalVisible := 'False'; ExternalWritable := 'False'; } AT MyWord : Array[0..15] of Bool;
      MyDInt { ExternalAccessible := 'False'; ExternalVisible := 'False'; ExternalWritable := 'False'; } : DInt;
      MyWordsinDint { ExternalAccessible := 'False'; ExternalVisible := 'False'; ExternalWritable := 'False'; } AT MyDInt : Array[0..1] of Word;
      MyReal { ExternalAccessible := 'False'; ExternalVisible := 'False'; ExternalWritable := 'False'; } : Real;
      MyWordsinReal { ExternalAccessible := 'False'; ExternalVisible := 'False'; ExternalWritable := 'False'; } AT MyReal : Array[0..1] of Word;
      MyInt { ExternalAccessible := 'False'; ExternalVisible := 'False'; ExternalWritable := 'False'; } : Int;
      MyWordinInt { ExternalAccessible := 'False'; ExternalVisible := 'False'; ExternalWritable := 'False'; } AT MyInt : Word;
      MyDWord { ExternalAccessible := 'False'; ExternalVisible := 'False'; ExternalWritable := 'False'; } : DWord;
      MyWordsinDWord { ExternalAccessible := 'False'; ExternalVisible := 'False'; ExternalWritable := 'False'; } AT MyDWord : Array[0..1] of Word;
      MyTime { ExternalAccessible := 'False'; ExternalVisible := 'False'; ExternalWritable := 'False'; } : Time;
      MyWordsinTime { ExternalAccessible := 'False'; ExternalVisible := 'False'; ExternalWritable := 'False'; } AT MyTime : Array[0..1] of Word;
      MyString { ExternalAccessible := 'False'; ExternalVisible := 'False'; ExternalWritable := 'False'; } : String[40];
      MyWordsinString { ExternalAccessible := 'False'; ExternalVisible := 'False'; ExternalWritable := 'False'; } AT MyString : Array[0..20] of Word;
   END_VAR
   VAR_TEMP
      HashModbus : DInt;
      HashIFA : DInt;
      HashTIAMap : DInt;
      i : Int;
   END_VAR
    //Author: Miklos Boros (miklos.boros@esss.se), Copyrigth 2017-2020 by European Spallation Source, Lund
    //This block was generated by PLCFactory, please don't change it MANUALLY!
    //Input File Name: Spk-000CDL_Cryo-PLC-010-template-IFA-20220922093722.ifa
    //Generated: 20220922093722
    //According to HASH: 457744924
    //Device type: ICS_LT
    //Description: This function does the variable mapping for a device. All device-variable will be linked to an interface variable defined in this block.

    //********************************************
    //****************HASH check******************
    //********************************************


    #MyWordsinDint[0] := "EPICSToPLC"."Word"[0];
    #MyWordsinDint[1] := "EPICSToPLC"."Word"[1];
    #HashModbus := #MyDInt; //Hash from EPICS/ModbusTCP

    #HashIFA := 457744924; //Hash from Interface Factory as a constant

    #MyWordsinDint[0] := "PLCToEPICS"."Word"[0];
    #MyWordsinDint[1] := "PLCToEPICS"."Word"[1];
    #HashTIAMap := #MyDInt; //Hash from PLCFactory TIA Map


    IF ((#HashIFA = #HashModbus) AND (#HashModbus = #HashTIAMap)) THEN //Check CRCs
        #DEVICE_PARAM_OK := TRUE;
       //##################################### ICS HWI ###############################################
       //############################  ICS Instrument Library     ####################################
       //#  PLC Sample Code in VersionDog: ICS_LIBRARY_MASTER_PLC                                   ##
       //#  CCDB device types: ICS_xxxxx                                                            ##
       //#  EPICS HMI (Block Icons/Faceplates)@ GitLab. Projekt: Cryo / CryogenicsLibrary / CryoLib ##
       //#                                                                                          ##
       //#                          LT- Level Transmitter in percent                                ##
       //#                                                                                          ##
       //#                                                                                          ##
       //###########################         Version: 1.4             ################################
       //Author:  Emilio Asensi
       //Date:    06-09-2022
       //Version: v1.4
       //Changes:
       //1. Added pvs for timer, filter and ramping speed
       //###########################         Version: 1.3             ################################
       //Author:  Miklos Boros
       //Date:    27-05-2019
       //Version: v1.3
       //Changes:
       //1. Variable Name Unification
       //###########################         Version: 1.2             ################################
       //Author:  Miklos Boros
       //Date:    28-02-2019
       //Version: v1.2
       //Changes:
       //1. Major review,
       //2. Indent,  unit standardization
       //###########################         Version: 1.1             ################################
       //Author:  Miklos Boros, Marino Vojneski
       //Date:    12-06-2018
       //Version: v1.1
       //Changes:
       //1. Modified Alarm Signal section to be compatible with new format.
       //########################### Version: 1.0             ########################################
       //Author:  Miklos Boros
       //Date:    25-01-2018
       //Version: v1.0
       //###########################
       //STATUS BLOCK
       //###########################
       //Operation modes
       //OPI buttons
       //Limits

    //********************************************
    //*************STATUS VARIABLES***************
    //********************************************


       #MyWord := W#0;
       #MyBoolsinWord[8] := #"OpMode_FreeRun";    //EPICSName: OpMode_FreeRun
       #MyBoolsinWord[9] := #"OpMode_Forced";    //EPICSName: OpMode_Forced
       #MyBoolsinWord[10] := #"Inhibit_Manual";    //EPICSName: Inhibit_Manual
       #MyBoolsinWord[11] := #"Inhibit_Force";    //EPICSName: Inhibit_Force
       #MyBoolsinWord[12] := #"Inhibit_Lock";    //EPICSName: Inhibit_Lock
       "PLCToEPICS"."Word"[#PLCToEPICSDataBlockOffset + 0] := #MyWord;

       #MyInt := #"TransmitterColor";    //EPICSName: TransmitterColor
       "PLCToEPICS"."Word"[#PLCToEPICSDataBlockOffset + 1] := #MyWordinInt;

       #MyWord := W#0;
       #MyBoolsinWord[8] := #"EnableFreeRunBtn";    //EPICSName: EnableFreeRunBtn
       #MyBoolsinWord[9] := #"EnableForcedBtn";    //EPICSName: EnableForcedBtn
       #MyBoolsinWord[10] := #"EnableManualBtn";    //EPICSName: EnableManualBtn
       "PLCToEPICS"."Word"[#PLCToEPICSDataBlockOffset + 2] := #MyWord;

       #MyReal := #"ScaleLOW";    //EPICSName: ScaleLOW
       "PLCToEPICS"."Word"[#PLCToEPICSDataBlockOffset + 3] := #MyWordsinReal[0];
       "PLCToEPICS"."Word"[#PLCToEPICSDataBlockOffset + 4] := #MyWordsinReal[1];

       #MyReal := #"ScaleHIGH";    //EPICSName: ScaleHIGH
       "PLCToEPICS"."Word"[#PLCToEPICSDataBlockOffset + 5] := #MyWordsinReal[0];
       "PLCToEPICS"."Word"[#PLCToEPICSDataBlockOffset + 6] := #MyWordsinReal[1];

       #MyReal := #"MeasValue";    //EPICSName: MeasValue
       "PLCToEPICS"."Word"[#PLCToEPICSDataBlockOffset + 7] := #MyWordsinReal[0];
       "PLCToEPICS"."Word"[#PLCToEPICSDataBlockOffset + 8] := #MyWordsinReal[1];

       #MyReal := #"RAWValue";    //EPICSName: RAWValue
       "PLCToEPICS"."Word"[#PLCToEPICSDataBlockOffset + 9] := #MyWordsinReal[0];
       "PLCToEPICS"."Word"[#PLCToEPICSDataBlockOffset + 10] := #MyWordsinReal[1];

       #MyWord := W#0;
       #MyBoolsinWord[8] := #"DevLocked";    //EPICSName: DevLocked
       "PLCToEPICS"."Word"[#PLCToEPICSDataBlockOffset + 11] := #MyWord;

       #MyDInt := #"Faceplate_LockID";    //EPICSName: Faceplate_LockID
       "PLCToEPICS"."Word"[#PLCToEPICSDataBlockOffset + 12] := #MyWordsinDint[0];
       "PLCToEPICS"."Word"[#PLCToEPICSDataBlockOffset + 13] := #MyWordsinDint[1];

       #MyDInt := #"BlockIcon_LockID";    //EPICSName: BlockIcon_LockID
       "PLCToEPICS"."Word"[#PLCToEPICSDataBlockOffset + 14] := #MyWordsinDint[0];
       "PLCToEPICS"."Word"[#PLCToEPICSDataBlockOffset + 15] := #MyWordsinDint[1];

       #MyWord := W#0;
       #MyBoolsinWord[8] := #"LatchAlarm";    //EPICSName: LatchAlarm
       #MyBoolsinWord[9] := #"GroupAlarm";    //EPICSName: GroupAlarm
       #MyBoolsinWord[10] := #"Underrange";    //EPICSName: Underrange
       #MyBoolsinWord[11] := #"Overrange";    //EPICSName: Overrange
       #MyBoolsinWord[12] := #"HIHI";    //EPICSName: HIHI
       #MyBoolsinWord[13] := #"HI";    //EPICSName: HI
       #MyBoolsinWord[14] := #"LO";    //EPICSName: LO
       #MyBoolsinWord[15] := #"LOLO";    //EPICSName: LOLO
       #MyBoolsinWord[0] := #"IO_Error";    //EPICSName: IO_Error
       #MyBoolsinWord[1] := #"Module_Error";    //EPICSName: Module_Error
       #MyBoolsinWord[2] := #"Param_Error";    //EPICSName: Param_Error
       "PLCToEPICS"."Word"[#PLCToEPICSDataBlockOffset + 16] := #MyWord;

       #MyReal := #"FB_ForceValue";    //EPICSName: FB_ForceValue
       "PLCToEPICS"."Word"[#PLCToEPICSDataBlockOffset + 17] := #MyWordsinReal[0];
       "PLCToEPICS"."Word"[#PLCToEPICSDataBlockOffset + 18] := #MyWordsinReal[1];

       #MyReal := #"FB_Limit_HIHI";    //EPICSName: FB_Limit_HIHI
       "PLCToEPICS"."Word"[#PLCToEPICSDataBlockOffset + 19] := #MyWordsinReal[0];
       "PLCToEPICS"."Word"[#PLCToEPICSDataBlockOffset + 20] := #MyWordsinReal[1];

       #MyReal := #"FB_Limit_HI";    //EPICSName: FB_Limit_HI
       "PLCToEPICS"."Word"[#PLCToEPICSDataBlockOffset + 21] := #MyWordsinReal[0];
       "PLCToEPICS"."Word"[#PLCToEPICSDataBlockOffset + 22] := #MyWordsinReal[1];

       #MyReal := #"FB_Limit_LO";    //EPICSName: FB_Limit_LO
       "PLCToEPICS"."Word"[#PLCToEPICSDataBlockOffset + 23] := #MyWordsinReal[0];
       "PLCToEPICS"."Word"[#PLCToEPICSDataBlockOffset + 24] := #MyWordsinReal[1];

       #MyReal := #"FB_Limit_LOLO";    //EPICSName: FB_Limit_LOLO
       "PLCToEPICS"."Word"[#PLCToEPICSDataBlockOffset + 25] := #MyWordsinReal[0];
       "PLCToEPICS"."Word"[#PLCToEPICSDataBlockOffset + 26] := #MyWordsinReal[1];

       #MyWord := W#0;
       #MyBoolsinWord[8] := #"Timer_enabled";    //EPICSName: Timer_enabled
       #MyBoolsinWord[9] := #"T_triggered";    //EPICSName: T_triggered
       "PLCToEPICS"."Word"[#PLCToEPICSDataBlockOffset + 27] := #MyWord;

       #MyInt := #"T_running";    //EPICSName: T_running
       "PLCToEPICS"."Word"[#PLCToEPICSDataBlockOffset + 28] := #MyWordinInt;

       #MyWord := W#0;
       #MyBoolsinWord[8] := #"F_enabled";    //EPICSName: F_enabled
       "PLCToEPICS"."Word"[#PLCToEPICSDataBlockOffset + 29] := #MyWord;

       #MyReal := #"FiltedValue";    //EPICSName: FiltedValue
       "PLCToEPICS"."Word"[#PLCToEPICSDataBlockOffset + 30] := #MyWordsinReal[0];
       "PLCToEPICS"."Word"[#PLCToEPICSDataBlockOffset + 31] := #MyWordsinReal[1];

    //********************************************
    //*************COMMAND VARIABLES**************
    //********************************************


       #MyWord := "EPICSToPLC"."Word"[#EPICSToPLCDataBlockOffset + 0];
       "EPICSToPLC"."Word"[#EPICSToPLCDataBlockOffset + 0] := 0;
       #"Cmd_FreeRun" := #MyBoolsinWord[8];    //EPICSName: Cmd_FreeRun
       #"Cmd_Force" := #MyBoolsinWord[9];    //EPICSName: Cmd_Force
       #"Cmd_ForceVal" := #MyBoolsinWord[10];    //EPICSName: Cmd_ForceVal
       #"Cmd_AckAlarm" := #MyBoolsinWord[11];    //EPICSName: Cmd_AckAlarm
       #"Cmd_ForceUnlock" := #MyBoolsinWord[12];    //EPICSName: Cmd_ForceUnlock
       #"Cmd_DevLock" := #MyBoolsinWord[13];    //EPICSName: Cmd_DevLock
       #"Cmd_DevUnlock" := #MyBoolsinWord[14];    //EPICSName: Cmd_DevUnlock

    //********************************************
    //************PARAMETER VARIABLES*************
    //********************************************


       #MyReal	:= 0.0;
       #MyWordsinReal[0]	:= "EPICSToPLC"."Word"[#EPICSToPLCDataBlockOffset + 1];
       #MyWordsinReal[1]	:= "EPICSToPLC"."Word"[#EPICSToPLCDataBlockOffset + 2];
       #"P_Limit_HIHI" := #MyReal;    //EPICSName: P_Limit_HIHI

       #MyReal	:= 0.0;
       #MyWordsinReal[0]	:= "EPICSToPLC"."Word"[#EPICSToPLCDataBlockOffset + 3];
       #MyWordsinReal[1]	:= "EPICSToPLC"."Word"[#EPICSToPLCDataBlockOffset + 4];
       #"P_Limit_HI" := #MyReal;    //EPICSName: P_Limit_HI

       #MyReal	:= 0.0;
       #MyWordsinReal[0]	:= "EPICSToPLC"."Word"[#EPICSToPLCDataBlockOffset + 5];
       #MyWordsinReal[1]	:= "EPICSToPLC"."Word"[#EPICSToPLCDataBlockOffset + 6];
       #"P_Limit_LO" := #MyReal;    //EPICSName: P_Limit_LO

       #MyReal	:= 0.0;
       #MyWordsinReal[0]	:= "EPICSToPLC"."Word"[#EPICSToPLCDataBlockOffset + 7];
       #MyWordsinReal[1]	:= "EPICSToPLC"."Word"[#EPICSToPLCDataBlockOffset + 8];
       #"P_Limit_LOLO" := #MyReal;    //EPICSName: P_Limit_LOLO

       #MyReal	:= 0.0;
       #MyWordsinReal[0]	:= "EPICSToPLC"."Word"[#EPICSToPLCDataBlockOffset + 9];
       #MyWordsinReal[1]	:= "EPICSToPLC"."Word"[#EPICSToPLCDataBlockOffset + 10];
       #"P_ForceValue" := #MyReal;    //EPICSName: P_ForceValue

       #MyDInt	:= 0;
       #MyWordsinDint[0]	:= "EPICSToPLC"."Word"[#EPICSToPLCDataBlockOffset + 11];
       #MyWordsinDint[1]	:= "EPICSToPLC"."Word"[#EPICSToPLCDataBlockOffset + 12];
       #"P_Faceplate_LockID" := #MyDInt;    //EPICSName: P_Faceplate_LockID

       #MyDInt	:= 0;
       #MyWordsinDint[0]	:= "EPICSToPLC"."Word"[#EPICSToPLCDataBlockOffset + 13];
       #MyWordsinDint[1]	:= "EPICSToPLC"."Word"[#EPICSToPLCDataBlockOffset + 14];
       #"P_BlockIcon_LockID" := #MyDInt;    //EPICSName: P_BlockIcon_LockID

       #MyWordinInt := "EPICSToPLC"."Word"[#EPICSToPLCDataBlockOffset + 15];
       #"T_period" := #MyInt;    //EPICSName: T_period

       #MyWordinInt := "EPICSToPLC"."Word"[#EPICSToPLCDataBlockOffset + 16];
       #"F_interval" := #MyInt;    //EPICSName: F_interval

       #MyWordinInt := "EPICSToPLC"."Word"[#EPICSToPLCDataBlockOffset + 17];
       #"F_buffer" := #MyInt;    //EPICSName: F_buffer

       #MyWord := "EPICSToPLC"."Word"[#EPICSToPLCDataBlockOffset + 18];
       #"F_Enable" := #MyBoolsinWord[8];    //EPICSName: F_Enable

       #MyReal	:= 0.0;
       #MyWordsinReal[0]	:= "EPICSToPLC"."Word"[#EPICSToPLCDataBlockOffset + 19];
       #MyWordsinReal[1]	:= "EPICSToPLC"."Word"[#EPICSToPLCDataBlockOffset + 20];
       #"P_RampUPSpeed" := #MyReal;    //EPICSName: P_RampUPSpeed

       #MyReal	:= 0.0;
       #MyWordsinReal[0]	:= "EPICSToPLC"."Word"[#EPICSToPLCDataBlockOffset + 21];
       #MyWordsinReal[1]	:= "EPICSToPLC"."Word"[#EPICSToPLCDataBlockOffset + 22];
       #"P_RampDNSpeed" := #MyReal;    //EPICSName: P_RampDNSpeed
    Else
       #DEVICE_PARAM_OK := FALSE; //Invalid Hash
    END_IF;
END_FUNCTION_BLOCK
FUNCTION_BLOCK "DEVTYPE_ICS_PT_mbar"
{ S7_Optimized_Access := 'TRUE' }
VERSION : 1.0
   VAR_INPUT
      "OpMode_FreeRun" { ExternalAccessible := 'True'; ExternalVisible := 'False'; ExternalWritable := 'False'; } : BOOL;   //EPICS Status variable: OpMode_FreeRun
      "OpMode_Forced" { ExternalAccessible := 'True'; ExternalVisible := 'False'; ExternalWritable := 'False'; } : BOOL;   //EPICS Status variable: OpMode_Forced
      "Inhibit_Manual" { ExternalAccessible := 'True'; ExternalVisible := 'False'; ExternalWritable := 'False'; } : BOOL;   //EPICS Status variable: Inhibit_Manual
      "Inhibit_Force" { ExternalAccessible := 'True'; ExternalVisible := 'False'; ExternalWritable := 'False'; } : BOOL;   //EPICS Status variable: Inhibit_Force
      "Inhibit_Lock" { ExternalAccessible := 'True'; ExternalVisible := 'False'; ExternalWritable := 'False'; } : BOOL;   //EPICS Status variable: Inhibit_Lock
      "TransmitterColor" { ExternalAccessible := 'True'; ExternalVisible := 'False'; ExternalWritable := 'False'; } : INT;   //EPICS Status variable: TransmitterColor
      "EnableFreeRunBtn" { ExternalAccessible := 'True'; ExternalVisible := 'False'; ExternalWritable := 'False'; } : BOOL;   //EPICS Status variable: EnableFreeRunBtn
      "EnableManualBtn" { ExternalAccessible := 'True'; ExternalVisible := 'False'; ExternalWritable := 'False'; } : BOOL;   //EPICS Status variable: EnableManualBtn
      "EnableForcedBtn" { ExternalAccessible := 'True'; ExternalVisible := 'False'; ExternalWritable := 'False'; } : BOOL;   //EPICS Status variable: EnableForcedBtn
      "ScaleLOW" { ExternalAccessible := 'True'; ExternalVisible := 'False'; ExternalWritable := 'False'; } : REAL;   //EPICS Status variable: ScaleLOW
      "ScaleHIGH" { ExternalAccessible := 'True'; ExternalVisible := 'False'; ExternalWritable := 'False'; } : REAL;   //EPICS Status variable: ScaleHIGH
      "MeasValue" { ExternalAccessible := 'True'; ExternalVisible := 'False'; ExternalWritable := 'False'; } : REAL;   //EPICS Status variable: MeasValue
      "DevLocked" { ExternalAccessible := 'True'; ExternalVisible := 'False'; ExternalWritable := 'False'; } : BOOL;   //EPICS Status variable: DevLocked
      "Faceplate_LockID" { ExternalAccessible := 'True'; ExternalVisible := 'False'; ExternalWritable := 'False'; } : DINT;   //EPICS Status variable: Faceplate_LockID
      "BlockIcon_LockID" { ExternalAccessible := 'True'; ExternalVisible := 'False'; ExternalWritable := 'False'; } : DINT;   //EPICS Status variable: BlockIcon_LockID
      "LatchAlarm" { ExternalAccessible := 'True'; ExternalVisible := 'False'; ExternalWritable := 'False'; } : BOOL;   //EPICS Status variable: LatchAlarm
      "GroupAlarm" { ExternalAccessible := 'True'; ExternalVisible := 'False'; ExternalWritable := 'False'; } : BOOL;   //EPICS Status variable: GroupAlarm
      "Underrange" { ExternalAccessible := 'True'; ExternalVisible := 'False'; ExternalWritable := 'False'; } : BOOL;   //EPICS Status variable: Underrange
      "Overrange" { ExternalAccessible := 'True'; ExternalVisible := 'False'; ExternalWritable := 'False'; } : BOOL;   //EPICS Status variable: Overrange
      "HIHI" { ExternalAccessible := 'True'; ExternalVisible := 'False'; ExternalWritable := 'False'; } : BOOL;   //EPICS Status variable: HIHI
      "HI" { ExternalAccessible := 'True'; ExternalVisible := 'False'; ExternalWritable := 'False'; } : BOOL;   //EPICS Status variable: HI
      "LO" { ExternalAccessible := 'True'; ExternalVisible := 'False'; ExternalWritable := 'False'; } : BOOL;   //EPICS Status variable: LO
      "LOLO" { ExternalAccessible := 'True'; ExternalVisible := 'False'; ExternalWritable := 'False'; } : BOOL;   //EPICS Status variable: LOLO
      "IO_Error" { ExternalAccessible := 'True'; ExternalVisible := 'False'; ExternalWritable := 'False'; } : BOOL;   //EPICS Status variable: IO_Error
      "Module_Error" { ExternalAccessible := 'True'; ExternalVisible := 'False'; ExternalWritable := 'False'; } : BOOL;   //EPICS Status variable: Module_Error
      "FB_ForceValue" { ExternalAccessible := 'True'; ExternalVisible := 'False'; ExternalWritable := 'False'; } : REAL;   //EPICS Status variable: FB_ForceValue
      "FB_Limit_HIHI" { ExternalAccessible := 'True'; ExternalVisible := 'False'; ExternalWritable := 'False'; } : REAL;   //EPICS Status variable: FB_Limit_HIHI
      "FB_Limit_HI" { ExternalAccessible := 'True'; ExternalVisible := 'False'; ExternalWritable := 'False'; } : REAL;   //EPICS Status variable: FB_Limit_HI
      "FB_Limit_LO" { ExternalAccessible := 'True'; ExternalVisible := 'False'; ExternalWritable := 'False'; } : REAL;   //EPICS Status variable: FB_Limit_LO
      "FB_Limit_LOLO" { ExternalAccessible := 'True'; ExternalVisible := 'False'; ExternalWritable := 'False'; } : REAL;   //EPICS Status variable: FB_Limit_LOLO
   EPICSToPLCLength { ExternalAccessible := 'False'; ExternalVisible := 'False'; ExternalWritable := 'False'; } : Int;   // Length of device command register array (in words)
   EPICSToPLCDataBlockOffset { ExternalAccessible := 'False'; ExternalVisible := 'False'; ExternalWritable := 'False'; } : Int;   // Offset in EPICS->PLC comms block where this device data resides (in words)
   PLCToEPICSLength { ExternalAccessible := 'False'; ExternalVisible := 'False'; ExternalWritable := 'False'; } : Int;   // Length of device status register array (in words)
   PLCToEPICSDataBlockOffset { ExternalAccessible := 'False'; ExternalVisible := 'False'; ExternalWritable := 'False'; } : Int;   // Offset in PLC->EPICS comms block where this device data resides (in words)
   END_VAR
   VAR_OUTPUT
      "Cmd_FreeRun" { ExternalAccessible := 'True'; ExternalVisible := 'False'; ExternalWritable := 'False'; } : BOOL;   //EPICS Command variable: Cmd_FreeRun
      "Cmd_Force" { ExternalAccessible := 'True'; ExternalVisible := 'False'; ExternalWritable := 'False'; } : BOOL;   //EPICS Command variable: Cmd_Force
      "Cmd_ForceVal" { ExternalAccessible := 'True'; ExternalVisible := 'False'; ExternalWritable := 'False'; } : BOOL;   //EPICS Command variable: Cmd_ForceVal
      "Cmd_AckAlarm" { ExternalAccessible := 'True'; ExternalVisible := 'False'; ExternalWritable := 'False'; } : BOOL;   //EPICS Command variable: Cmd_AckAlarm
      "Cmd_ForceUnlock" { ExternalAccessible := 'True'; ExternalVisible := 'False'; ExternalWritable := 'False'; } : BOOL;   //EPICS Command variable: Cmd_ForceUnlock
      "Cmd_DevLock" { ExternalAccessible := 'True'; ExternalVisible := 'False'; ExternalWritable := 'False'; } : BOOL;   //EPICS Command variable: Cmd_DevLock
      "Cmd_DevUnlock" { ExternalAccessible := 'True'; ExternalVisible := 'False'; ExternalWritable := 'False'; } : BOOL;   //EPICS Command variable: Cmd_DevUnlock
      "P_Limit_HIHI" { ExternalAccessible := 'True'; ExternalVisible := 'False'; ExternalWritable := 'False'; } : REAL;   //EPICS Parameter variable: P_Limit_HIHI
      "P_Limit_HI" { ExternalAccessible := 'True'; ExternalVisible := 'False'; ExternalWritable := 'False'; } : REAL;   //EPICS Parameter variable: P_Limit_HI
      "P_Limit_LO" { ExternalAccessible := 'True'; ExternalVisible := 'False'; ExternalWritable := 'False'; } : REAL;   //EPICS Parameter variable: P_Limit_LO
      "P_Limit_LOLO" { ExternalAccessible := 'True'; ExternalVisible := 'False'; ExternalWritable := 'False'; } : REAL;   //EPICS Parameter variable: P_Limit_LOLO
      "P_ForceValue" { ExternalAccessible := 'True'; ExternalVisible := 'False'; ExternalWritable := 'False'; } : REAL;   //EPICS Parameter variable: P_ForceValue
      "P_Faceplate_LockID" { ExternalAccessible := 'True'; ExternalVisible := 'False'; ExternalWritable := 'False'; } : DINT;   //EPICS Parameter variable: P_Faceplate_LockID
      "P_BlockIcon_LockID" { ExternalAccessible := 'True'; ExternalVisible := 'False'; ExternalWritable := 'False'; } : DINT;   //EPICS Parameter variable: P_BlockIcon_LockID
      DEVICE_PARAM_OK { ExternalAccessible := 'False'; ExternalVisible := 'False'; ExternalWritable := 'False'; } : Bool;
   END_VAR
   VAR_IN_OUT
   END_VAR
   Var DB_SPECIFIC
      MyWord { ExternalAccessible := 'False'; ExternalVisible := 'False'; ExternalWritable := 'False'; } : Word;
      MyBytesinWord { ExternalAccessible := 'False'; ExternalVisible := 'False'; ExternalWritable := 'False'; } AT MyWord : Array[0..1] of Byte;
      MyBoolsinWord { ExternalAccessible := 'False'; ExternalVisible := 'False'; ExternalWritable := 'False'; } AT MyWord : Array[0..15] of Bool;
      MyDInt { ExternalAccessible := 'False'; ExternalVisible := 'False'; ExternalWritable := 'False'; } : DInt;
      MyWordsinDint { ExternalAccessible := 'False'; ExternalVisible := 'False'; ExternalWritable := 'False'; } AT MyDInt : Array[0..1] of Word;
      MyReal { ExternalAccessible := 'False'; ExternalVisible := 'False'; ExternalWritable := 'False'; } : Real;
      MyWordsinReal { ExternalAccessible := 'False'; ExternalVisible := 'False'; ExternalWritable := 'False'; } AT MyReal : Array[0..1] of Word;
      MyInt { ExternalAccessible := 'False'; ExternalVisible := 'False'; ExternalWritable := 'False'; } : Int;
      MyWordinInt { ExternalAccessible := 'False'; ExternalVisible := 'False'; ExternalWritable := 'False'; } AT MyInt : Word;
      MyDWord { ExternalAccessible := 'False'; ExternalVisible := 'False'; ExternalWritable := 'False'; } : DWord;
      MyWordsinDWord { ExternalAccessible := 'False'; ExternalVisible := 'False'; ExternalWritable := 'False'; } AT MyDWord : Array[0..1] of Word;
      MyTime { ExternalAccessible := 'False'; ExternalVisible := 'False'; ExternalWritable := 'False'; } : Time;
      MyWordsinTime { ExternalAccessible := 'False'; ExternalVisible := 'False'; ExternalWritable := 'False'; } AT MyTime : Array[0..1] of Word;
      MyString { ExternalAccessible := 'False'; ExternalVisible := 'False'; ExternalWritable := 'False'; } : String[40];
      MyWordsinString { ExternalAccessible := 'False'; ExternalVisible := 'False'; ExternalWritable := 'False'; } AT MyString : Array[0..20] of Word;
   END_VAR
   VAR_TEMP
      HashModbus : DInt;
      HashIFA : DInt;
      HashTIAMap : DInt;
      i : Int;
   END_VAR
    //Author: Miklos Boros (miklos.boros@esss.se), Copyrigth 2017-2020 by European Spallation Source, Lund
    //This block was generated by PLCFactory, please don't change it MANUALLY!
    //Input File Name: Spk-000CDL_Cryo-PLC-010-template-IFA-20220922093722.ifa
    //Generated: 20220922093722
    //According to HASH: 457744924
    //Device type: ICS_PT_mbar
    //Description: This function does the variable mapping for a device. All device-variable will be linked to an interface variable defined in this block.

    //********************************************
    //****************HASH check******************
    //********************************************


    #MyWordsinDint[0] := "EPICSToPLC"."Word"[0];
    #MyWordsinDint[1] := "EPICSToPLC"."Word"[1];
    #HashModbus := #MyDInt; //Hash from EPICS/ModbusTCP

    #HashIFA := 457744924; //Hash from Interface Factory as a constant

    #MyWordsinDint[0] := "PLCToEPICS"."Word"[0];
    #MyWordsinDint[1] := "PLCToEPICS"."Word"[1];
    #HashTIAMap := #MyDInt; //Hash from PLCFactory TIA Map


    IF ((#HashIFA = #HashModbus) AND (#HashModbus = #HashTIAMap)) THEN //Check CRCs
        #DEVICE_PARAM_OK := TRUE;
       //##################################### ICS HWI ###############################################
       //############################  ICS Instrument Library     ####################################
       //#  PLC Sample Code in VersionDog: ICS_LIBRARY_MASTER_PLC                                   ##
       //#  CCDB device types: ICS_xxxxx                                                            ##
       //#  EPICS HMI (Block Icons/Faceplates)@ GitLab. Projekt: Cryo / CryogenicsLibrary / CryoLib ##
       //#                                                                                          ##
       //#                             PT - Pressure Transmitter in mbar                            ##
       //#                                                                                          ##
       //#                                                                                          ##
       //###########################         Version: 1.3             ################################
       //Author:  Miklos Boros
       //Date:    27-05-2019
       //Version: v1.3
       //Changes:
       //1. Variable Name Unification
       //###########################         Version: 1.2             ################################
       //Author:  Miklos Boros
       //Date:    28-02-2019
       //Version: v1.2
       //Changes:
       //1. Major review,
       //2. Indent,  unit standardization
       //###########################         Version: 1.1             ################################
       //Author:  Miklos Boros, Marino Vojneski
       //Date:    12-06-2018
       //Version: v1.1
       //Changes:
       //1. Modified Alarm Signal section to be compatible with new format.
       //########################### Version: 1.0             ########################################
       //Author:  Miklos Boros
       //Date:    25-01-2018
       //Version: v1.0
       //###########################
       //STATUS BLOCK
       //###########################
       //Operation modes
       //OPI buttons
       //Limits

    //********************************************
    //*************STATUS VARIABLES***************
    //********************************************


       #MyWord := W#0;
       #MyBoolsinWord[8] := #"OpMode_FreeRun";    //EPICSName: OpMode_FreeRun
       #MyBoolsinWord[9] := #"OpMode_Forced";    //EPICSName: OpMode_Forced
       #MyBoolsinWord[10] := #"Inhibit_Manual";    //EPICSName: Inhibit_Manual
       #MyBoolsinWord[11] := #"Inhibit_Force";    //EPICSName: Inhibit_Force
       #MyBoolsinWord[12] := #"Inhibit_Lock";    //EPICSName: Inhibit_Lock
       "PLCToEPICS"."Word"[#PLCToEPICSDataBlockOffset + 0] := #MyWord;

       #MyInt := #"TransmitterColor";    //EPICSName: TransmitterColor
       "PLCToEPICS"."Word"[#PLCToEPICSDataBlockOffset + 1] := #MyWordinInt;

       #MyWord := W#0;
       #MyBoolsinWord[8] := #"EnableFreeRunBtn";    //EPICSName: EnableFreeRunBtn
       #MyBoolsinWord[9] := #"EnableManualBtn";    //EPICSName: EnableManualBtn
       #MyBoolsinWord[10] := #"EnableForcedBtn";    //EPICSName: EnableForcedBtn
       "PLCToEPICS"."Word"[#PLCToEPICSDataBlockOffset + 2] := #MyWord;

       #MyReal := #"ScaleLOW";    //EPICSName: ScaleLOW
       "PLCToEPICS"."Word"[#PLCToEPICSDataBlockOffset + 3] := #MyWordsinReal[0];
       "PLCToEPICS"."Word"[#PLCToEPICSDataBlockOffset + 4] := #MyWordsinReal[1];

       #MyReal := #"ScaleHIGH";    //EPICSName: ScaleHIGH
       "PLCToEPICS"."Word"[#PLCToEPICSDataBlockOffset + 5] := #MyWordsinReal[0];
       "PLCToEPICS"."Word"[#PLCToEPICSDataBlockOffset + 6] := #MyWordsinReal[1];

       #MyReal := #"MeasValue";    //EPICSName: MeasValue
       "PLCToEPICS"."Word"[#PLCToEPICSDataBlockOffset + 7] := #MyWordsinReal[0];
       "PLCToEPICS"."Word"[#PLCToEPICSDataBlockOffset + 8] := #MyWordsinReal[1];

       #MyWord := W#0;
       #MyBoolsinWord[8] := #"DevLocked";    //EPICSName: DevLocked
       "PLCToEPICS"."Word"[#PLCToEPICSDataBlockOffset + 9] := #MyWord;

       #MyDInt := #"Faceplate_LockID";    //EPICSName: Faceplate_LockID
       "PLCToEPICS"."Word"[#PLCToEPICSDataBlockOffset + 10] := #MyWordsinDint[0];
       "PLCToEPICS"."Word"[#PLCToEPICSDataBlockOffset + 11] := #MyWordsinDint[1];

       #MyDInt := #"BlockIcon_LockID";    //EPICSName: BlockIcon_LockID
       "PLCToEPICS"."Word"[#PLCToEPICSDataBlockOffset + 12] := #MyWordsinDint[0];
       "PLCToEPICS"."Word"[#PLCToEPICSDataBlockOffset + 13] := #MyWordsinDint[1];

       #MyWord := W#0;
       #MyBoolsinWord[8] := #"LatchAlarm";    //EPICSName: LatchAlarm
       #MyBoolsinWord[9] := #"GroupAlarm";    //EPICSName: GroupAlarm
       #MyBoolsinWord[10] := #"Underrange";    //EPICSName: Underrange
       #MyBoolsinWord[11] := #"Overrange";    //EPICSName: Overrange
       #MyBoolsinWord[12] := #"HIHI";    //EPICSName: HIHI
       #MyBoolsinWord[13] := #"HI";    //EPICSName: HI
       #MyBoolsinWord[14] := #"LO";    //EPICSName: LO
       #MyBoolsinWord[15] := #"LOLO";    //EPICSName: LOLO
       #MyBoolsinWord[0] := #"IO_Error";    //EPICSName: IO_Error
       #MyBoolsinWord[1] := #"Module_Error";    //EPICSName: Module_Error
       "PLCToEPICS"."Word"[#PLCToEPICSDataBlockOffset + 14] := #MyWord;

       #MyReal := #"FB_ForceValue";    //EPICSName: FB_ForceValue
       "PLCToEPICS"."Word"[#PLCToEPICSDataBlockOffset + 15] := #MyWordsinReal[0];
       "PLCToEPICS"."Word"[#PLCToEPICSDataBlockOffset + 16] := #MyWordsinReal[1];

       #MyReal := #"FB_Limit_HIHI";    //EPICSName: FB_Limit_HIHI
       "PLCToEPICS"."Word"[#PLCToEPICSDataBlockOffset + 17] := #MyWordsinReal[0];
       "PLCToEPICS"."Word"[#PLCToEPICSDataBlockOffset + 18] := #MyWordsinReal[1];

       #MyReal := #"FB_Limit_HI";    //EPICSName: FB_Limit_HI
       "PLCToEPICS"."Word"[#PLCToEPICSDataBlockOffset + 19] := #MyWordsinReal[0];
       "PLCToEPICS"."Word"[#PLCToEPICSDataBlockOffset + 20] := #MyWordsinReal[1];

       #MyReal := #"FB_Limit_LO";    //EPICSName: FB_Limit_LO
       "PLCToEPICS"."Word"[#PLCToEPICSDataBlockOffset + 21] := #MyWordsinReal[0];
       "PLCToEPICS"."Word"[#PLCToEPICSDataBlockOffset + 22] := #MyWordsinReal[1];

       #MyReal := #"FB_Limit_LOLO";    //EPICSName: FB_Limit_LOLO
       "PLCToEPICS"."Word"[#PLCToEPICSDataBlockOffset + 23] := #MyWordsinReal[0];
       "PLCToEPICS"."Word"[#PLCToEPICSDataBlockOffset + 24] := #MyWordsinReal[1];

    //********************************************
    //*************COMMAND VARIABLES**************
    //********************************************


       #MyWord := "EPICSToPLC"."Word"[#EPICSToPLCDataBlockOffset + 0];
       "EPICSToPLC"."Word"[#EPICSToPLCDataBlockOffset + 0] := 0;
       #"Cmd_FreeRun" := #MyBoolsinWord[8];    //EPICSName: Cmd_FreeRun
       #"Cmd_Force" := #MyBoolsinWord[9];    //EPICSName: Cmd_Force
       #"Cmd_ForceVal" := #MyBoolsinWord[10];    //EPICSName: Cmd_ForceVal
       #"Cmd_AckAlarm" := #MyBoolsinWord[11];    //EPICSName: Cmd_AckAlarm
       #"Cmd_ForceUnlock" := #MyBoolsinWord[12];    //EPICSName: Cmd_ForceUnlock
       #"Cmd_DevLock" := #MyBoolsinWord[13];    //EPICSName: Cmd_DevLock
       #"Cmd_DevUnlock" := #MyBoolsinWord[14];    //EPICSName: Cmd_DevUnlock

    //********************************************
    //************PARAMETER VARIABLES*************
    //********************************************


       #MyReal	:= 0.0;
       #MyWordsinReal[0]	:= "EPICSToPLC"."Word"[#EPICSToPLCDataBlockOffset + 1];
       #MyWordsinReal[1]	:= "EPICSToPLC"."Word"[#EPICSToPLCDataBlockOffset + 2];
       #"P_Limit_HIHI" := #MyReal;    //EPICSName: P_Limit_HIHI

       #MyReal	:= 0.0;
       #MyWordsinReal[0]	:= "EPICSToPLC"."Word"[#EPICSToPLCDataBlockOffset + 3];
       #MyWordsinReal[1]	:= "EPICSToPLC"."Word"[#EPICSToPLCDataBlockOffset + 4];
       #"P_Limit_HI" := #MyReal;    //EPICSName: P_Limit_HI

       #MyReal	:= 0.0;
       #MyWordsinReal[0]	:= "EPICSToPLC"."Word"[#EPICSToPLCDataBlockOffset + 5];
       #MyWordsinReal[1]	:= "EPICSToPLC"."Word"[#EPICSToPLCDataBlockOffset + 6];
       #"P_Limit_LO" := #MyReal;    //EPICSName: P_Limit_LO

       #MyReal	:= 0.0;
       #MyWordsinReal[0]	:= "EPICSToPLC"."Word"[#EPICSToPLCDataBlockOffset + 7];
       #MyWordsinReal[1]	:= "EPICSToPLC"."Word"[#EPICSToPLCDataBlockOffset + 8];
       #"P_Limit_LOLO" := #MyReal;    //EPICSName: P_Limit_LOLO

       #MyReal	:= 0.0;
       #MyWordsinReal[0]	:= "EPICSToPLC"."Word"[#EPICSToPLCDataBlockOffset + 9];
       #MyWordsinReal[1]	:= "EPICSToPLC"."Word"[#EPICSToPLCDataBlockOffset + 10];
       #"P_ForceValue" := #MyReal;    //EPICSName: P_ForceValue

       #MyDInt	:= 0;
       #MyWordsinDint[0]	:= "EPICSToPLC"."Word"[#EPICSToPLCDataBlockOffset + 11];
       #MyWordsinDint[1]	:= "EPICSToPLC"."Word"[#EPICSToPLCDataBlockOffset + 12];
       #"P_Faceplate_LockID" := #MyDInt;    //EPICSName: P_Faceplate_LockID

       #MyDInt	:= 0;
       #MyWordsinDint[0]	:= "EPICSToPLC"."Word"[#EPICSToPLCDataBlockOffset + 13];
       #MyWordsinDint[1]	:= "EPICSToPLC"."Word"[#EPICSToPLCDataBlockOffset + 14];
       #"P_BlockIcon_LockID" := #MyDInt;    //EPICSName: P_BlockIcon_LockID
    Else
       #DEVICE_PARAM_OK := FALSE; //Invalid Hash
    END_IF;
END_FUNCTION_BLOCK

DATA_BLOCK "DEV_Spk-000CDL:SC-FSM-300_iDB"
{ S7_Optimized_Access := 'TRUE' }
VERSION : 1.0
NON_RETAIN
"DEVTYPE_C3S_AUTO_CONF"
BEGIN
END_DATA_BLOCK


DATA_BLOCK "DEV_Spk-000CDL:SC-FSM-400_iDB"
{ S7_Optimized_Access := 'TRUE' }
VERSION : 1.0
NON_RETAIN
"DEVTYPE_C3S_DIAG"
BEGIN
END_DATA_BLOCK


DATA_BLOCK "DEV_Spk-000CDL:SC-FSM-500_iDB"
{ S7_Optimized_Access := 'TRUE' }
VERSION : 1.0
NON_RETAIN
"DEVTYPE_C3S_INTLCK"
BEGIN
END_DATA_BLOCK


DATA_BLOCK "DEV_Spk-000CDL:SC-FSM-600_iDB"
{ S7_Optimized_Access := 'TRUE' }
VERSION : 1.0
NON_RETAIN
"DEVTYPE_C3S_MODE_SEL"
BEGIN
END_DATA_BLOCK


DATA_BLOCK "DEV_Spk-000CDL:Cryo-PID-91_iDB"
{ S7_Optimized_Access := 'TRUE' }
VERSION : 1.0
NON_RETAIN
"DEVTYPE_C3S_PID"
BEGIN
END_DATA_BLOCK


DATA_BLOCK "DEV_Spk-000CDL:Cryo-PID-92_iDB"
{ S7_Optimized_Access := 'TRUE' }
VERSION : 1.0
NON_RETAIN
"DEVTYPE_C3S_PID"
BEGIN
END_DATA_BLOCK


DATA_BLOCK "DEV_Spk-000CDL:Cryo-PID-93_iDB"
{ S7_Optimized_Access := 'TRUE' }
VERSION : 1.0
NON_RETAIN
"DEVTYPE_C3S_PID"
BEGIN
END_DATA_BLOCK


DATA_BLOCK "DEV_Spk-000CDL:Cryo-PID-94_iDB"
{ S7_Optimized_Access := 'TRUE' }
VERSION : 1.0
NON_RETAIN
"DEVTYPE_C3S_PID"
BEGIN
END_DATA_BLOCK


DATA_BLOCK "DEV_Spk-000CDL:Cryo-CV-91_iDB"
{ S7_Optimized_Access := 'TRUE' }
VERSION : 1.0
NON_RETAIN
"DEVTYPE_ICS_CV_PB_SIPART"
BEGIN
END_DATA_BLOCK


DATA_BLOCK "DEV_Spk-000CDL:Cryo-CV-92_iDB"
{ S7_Optimized_Access := 'TRUE' }
VERSION : 1.0
NON_RETAIN
"DEVTYPE_ICS_CV_PB_SIPART"
BEGIN
END_DATA_BLOCK


DATA_BLOCK "DEV_Spk-000CDL:Cryo-CV-93_iDB"
{ S7_Optimized_Access := 'TRUE' }
VERSION : 1.0
NON_RETAIN
"DEVTYPE_ICS_CV_PB_SIPART"
BEGIN
END_DATA_BLOCK


DATA_BLOCK "DEV_Spk-000CDL:Cryo-CV-94_iDB"
{ S7_Optimized_Access := 'TRUE' }
VERSION : 1.0
NON_RETAIN
"DEVTYPE_ICS_CV_PB_SIPART"
BEGIN
END_DATA_BLOCK


DATA_BLOCK "DEV_Spk-000CDL:Cryo-EH-91_iDB"
{ S7_Optimized_Access := 'TRUE' }
VERSION : 1.0
NON_RETAIN
"DEVTYPE_ICS_EH"
BEGIN
END_DATA_BLOCK


DATA_BLOCK "DEV_Spk-000CDL:Cryo-EH-92_iDB"
{ S7_Optimized_Access := 'TRUE' }
VERSION : 1.0
NON_RETAIN
"DEVTYPE_ICS_EH"
BEGIN
END_DATA_BLOCK


DATA_BLOCK "DEV_Spk-000CDL:Cryo-EH-93_iDB"
{ S7_Optimized_Access := 'TRUE' }
VERSION : 1.0
NON_RETAIN
"DEVTYPE_ICS_EH"
BEGIN
END_DATA_BLOCK


DATA_BLOCK "DEV_Spk-000CDL:Cryo-EH-94_iDB"
{ S7_Optimized_Access := 'TRUE' }
VERSION : 1.0
NON_RETAIN
"DEVTYPE_ICS_EH"
BEGIN
END_DATA_BLOCK


DATA_BLOCK "DEV_Spk-000CDL:Cryo-EH-95_iDB"
{ S7_Optimized_Access := 'TRUE' }
VERSION : 1.0
NON_RETAIN
"DEVTYPE_ICS_EH"
BEGIN
END_DATA_BLOCK


DATA_BLOCK "DEV_Spk-000CDL:Cryo-EH-96_iDB"
{ S7_Optimized_Access := 'TRUE' }
VERSION : 1.0
NON_RETAIN
"DEVTYPE_ICS_EH"
BEGIN
END_DATA_BLOCK


DATA_BLOCK "DEV_Spk-000CDL:Cryo-HV-70_iDB"
{ S7_Optimized_Access := 'TRUE' }
VERSION : 1.0
NON_RETAIN
"DEVTYPE_ICS_HV"
BEGIN
END_DATA_BLOCK


DATA_BLOCK "DEV_Spk-000CDL:Cryo-HV-73_iDB"
{ S7_Optimized_Access := 'TRUE' }
VERSION : 1.0
NON_RETAIN
"DEVTYPE_ICS_HV"
BEGIN
END_DATA_BLOCK


DATA_BLOCK "DEV_Spk-000CDL:Cryo-TT-91_iDB"
{ S7_Optimized_Access := 'TRUE' }
VERSION : 1.0
NON_RETAIN
"DEVTYPE_ICS_LAKESHORE_TT"
BEGIN
END_DATA_BLOCK


DATA_BLOCK "DEV_Spk-000CDL:Cryo-TT-92_iDB"
{ S7_Optimized_Access := 'TRUE' }
VERSION : 1.0
NON_RETAIN
"DEVTYPE_ICS_LAKESHORE_TT"
BEGIN
END_DATA_BLOCK


DATA_BLOCK "DEV_Spk-000CDL:Cryo-TT-93_iDB"
{ S7_Optimized_Access := 'TRUE' }
VERSION : 1.0
NON_RETAIN
"DEVTYPE_ICS_LAKESHORE_TT"
BEGIN
END_DATA_BLOCK


DATA_BLOCK "DEV_Spk-000CDL:Cryo-TT-94_iDB"
{ S7_Optimized_Access := 'TRUE' }
VERSION : 1.0
NON_RETAIN
"DEVTYPE_ICS_LAKESHORE_TT"
BEGIN
END_DATA_BLOCK


DATA_BLOCK "DEV_Spk-000CDL:Cryo-TT-95_iDB"
{ S7_Optimized_Access := 'TRUE' }
VERSION : 1.0
NON_RETAIN
"DEVTYPE_ICS_LAKESHORE_TT"
BEGIN
END_DATA_BLOCK


DATA_BLOCK "DEV_Spk-000CDL:Cryo-TT-96_iDB"
{ S7_Optimized_Access := 'TRUE' }
VERSION : 1.0
NON_RETAIN
"DEVTYPE_ICS_LAKESHORE_TT"
BEGIN
END_DATA_BLOCK


DATA_BLOCK "DEV_Spk-000CDL:Cryo-TT-97_iDB"
{ S7_Optimized_Access := 'TRUE' }
VERSION : 1.0
NON_RETAIN
"DEVTYPE_ICS_LAKESHORE_TT"
BEGIN
END_DATA_BLOCK


DATA_BLOCK "DEV_Spk-000CDL:Cryo-TT-98_iDB"
{ S7_Optimized_Access := 'TRUE' }
VERSION : 1.0
NON_RETAIN
"DEVTYPE_ICS_LAKESHORE_TT"
BEGIN
END_DATA_BLOCK


DATA_BLOCK "DEV_Spk-000CDL:Cryo-LT-91_iDB"
{ S7_Optimized_Access := 'TRUE' }
VERSION : 1.0
NON_RETAIN
"DEVTYPE_ICS_LT"
BEGIN
END_DATA_BLOCK


DATA_BLOCK "DEV_Spk-000CDL:Cryo-LT-92_iDB"
{ S7_Optimized_Access := 'TRUE' }
VERSION : 1.0
NON_RETAIN
"DEVTYPE_ICS_LT"
BEGIN
END_DATA_BLOCK


DATA_BLOCK "DEV_Spk-000CDL:Cryo-PT-91_iDB"
{ S7_Optimized_Access := 'TRUE' }
VERSION : 1.0
NON_RETAIN
"DEVTYPE_ICS_PT_mbar"
BEGIN
END_DATA_BLOCK


DATA_BLOCK "DEV_Spk-000CDL:Cryo-PT-92_iDB"
{ S7_Optimized_Access := 'TRUE' }
VERSION : 1.0
NON_RETAIN
"DEVTYPE_ICS_PT_mbar"
BEGIN
END_DATA_BLOCK


DATA_BLOCK "DEV_Spk-000CDL:Cryo-PT-93_iDB"
{ S7_Optimized_Access := 'TRUE' }
VERSION : 1.0
NON_RETAIN
"DEVTYPE_ICS_PT_mbar"
BEGIN
END_DATA_BLOCK


DATA_BLOCK "DEV_Spk-000CDL:Cryo-PT-94_iDB"
{ S7_Optimized_Access := 'TRUE' }
VERSION : 1.0
NON_RETAIN
"DEVTYPE_ICS_PT_mbar"
BEGIN
END_DATA_BLOCK


DATA_BLOCK "DEV_Spk-000CDL:Cryo-PT-95_iDB"
{ S7_Optimized_Access := 'TRUE' }
VERSION : 1.0
NON_RETAIN
"DEVTYPE_ICS_PT_mbar"
BEGIN
END_DATA_BLOCK


DATA_BLOCK "DEV_Spk-000CDL:Vac-VGC-071_iDB"
{ S7_Optimized_Access := 'TRUE' }
VERSION : 1.0
NON_RETAIN
"DEVTYPE_ICS_PT_mbar"
BEGIN
END_DATA_BLOCK


DATA_BLOCK "DEV_Spk-000CDL:Vac-VGP-070_iDB"
{ S7_Optimized_Access := 'TRUE' }
VERSION : 1.0
NON_RETAIN
"DEVTYPE_ICS_PT_mbar"
BEGIN
END_DATA_BLOCK

FUNCTION "EPICS_device_calls" : Void
{ S7_Optimized_Access := 'TRUE' }
VERSION : 1.0

   VAR_TEMP
      "Spk-000CDL:SC-FSM-300" : Bool;   // HASH codes are OK
      "Spk-000CDL:SC-FSM-400" : Bool;   // HASH codes are OK
      "Spk-000CDL:SC-FSM-500" : Bool;   // HASH codes are OK
      "Spk-000CDL:SC-FSM-600" : Bool;   // HASH codes are OK
      "Spk-000CDL:Cryo-PID-91" : Bool;   // HASH codes are OK
      "Spk-000CDL:Cryo-PID-92" : Bool;   // HASH codes are OK
      "Spk-000CDL:Cryo-PID-93" : Bool;   // HASH codes are OK
      "Spk-000CDL:Cryo-PID-94" : Bool;   // HASH codes are OK
      "Spk-000CDL:Cryo-CV-91" : Bool;   // HASH codes are OK
      "Spk-000CDL:Cryo-CV-92" : Bool;   // HASH codes are OK
      "Spk-000CDL:Cryo-CV-93" : Bool;   // HASH codes are OK
      "Spk-000CDL:Cryo-CV-94" : Bool;   // HASH codes are OK
      "Spk-000CDL:Cryo-EH-91" : Bool;   // HASH codes are OK
      "Spk-000CDL:Cryo-EH-92" : Bool;   // HASH codes are OK
      "Spk-000CDL:Cryo-EH-93" : Bool;   // HASH codes are OK
      "Spk-000CDL:Cryo-EH-94" : Bool;   // HASH codes are OK
      "Spk-000CDL:Cryo-EH-95" : Bool;   // HASH codes are OK
      "Spk-000CDL:Cryo-EH-96" : Bool;   // HASH codes are OK
      "Spk-000CDL:Cryo-HV-70" : Bool;   // HASH codes are OK
      "Spk-000CDL:Cryo-HV-73" : Bool;   // HASH codes are OK
      "Spk-000CDL:Cryo-TT-91" : Bool;   // HASH codes are OK
      "Spk-000CDL:Cryo-TT-92" : Bool;   // HASH codes are OK
      "Spk-000CDL:Cryo-TT-93" : Bool;   // HASH codes are OK
      "Spk-000CDL:Cryo-TT-94" : Bool;   // HASH codes are OK
      "Spk-000CDL:Cryo-TT-95" : Bool;   // HASH codes are OK
      "Spk-000CDL:Cryo-TT-96" : Bool;   // HASH codes are OK
      "Spk-000CDL:Cryo-TT-97" : Bool;   // HASH codes are OK
      "Spk-000CDL:Cryo-TT-98" : Bool;   // HASH codes are OK
      "Spk-000CDL:Cryo-LT-91" : Bool;   // HASH codes are OK
      "Spk-000CDL:Cryo-LT-92" : Bool;   // HASH codes are OK
      "Spk-000CDL:Cryo-PT-91" : Bool;   // HASH codes are OK
      "Spk-000CDL:Cryo-PT-92" : Bool;   // HASH codes are OK
      "Spk-000CDL:Cryo-PT-93" : Bool;   // HASH codes are OK
      "Spk-000CDL:Cryo-PT-94" : Bool;   // HASH codes are OK
      "Spk-000CDL:Cryo-PT-95" : Bool;   // HASH codes are OK
      "Spk-000CDL:Vac-VGC-071" : Bool;   // HASH codes are OK
      "Spk-000CDL:Vac-VGP-070" : Bool;   // HASH codes are OK
   END_VAR

BEGIN
      //Author: Miklos Boros (miklos.boros@esss.se), Copyrigth 2017-2020 by European Spallation Source, Lund
      //This block was generated by PLCFactory
      //According to HASH:457744924
      //Description: Description: This function calls the devices according to the corresponding device type

        //DO NOT Modify the following line!!!
        "Utilities".TestInProgress := FALSE;
        "Utilities".EPICS_Device_calls_precessed := TRUE;


        //********************************************
        // Device name: Spk-000CDL:SC-FSM-300
        // Device type: C3S_AUTO_CONF
        //********************************************

      "DEV_Spk-000CDL:SC-FSM-300_iDB" (EPICSToPLCLength:=73,
      EPICSToPLCDataBlockOffset:=10,
      PLCToEPICSLength:=73,
      PLCToEPICSDataBlockOffset:=10);

        //********************************************
        // Device name: Spk-000CDL:SC-FSM-400
        // Device type: C3S_DIAG
        //********************************************

      "DEV_Spk-000CDL:SC-FSM-400_iDB" (EPICSToPLCLength:=1,
      EPICSToPLCDataBlockOffset:=83,
      PLCToEPICSLength:=8,
      PLCToEPICSDataBlockOffset:=83);

        //********************************************
        // Device name: Spk-000CDL:SC-FSM-500
        // Device type: C3S_INTLCK
        //********************************************

      "DEV_Spk-000CDL:SC-FSM-500_iDB" (EPICSToPLCLength:=1,
      EPICSToPLCDataBlockOffset:=84,
      PLCToEPICSLength:=1,
      PLCToEPICSDataBlockOffset:=91);

        //********************************************
        // Device name: Spk-000CDL:SC-FSM-600
        // Device type: C3S_MODE_SEL
        //********************************************

      "DEV_Spk-000CDL:SC-FSM-600_iDB" (EPICSToPLCLength:=1,
      EPICSToPLCDataBlockOffset:=85,
      PLCToEPICSLength:=25,
      PLCToEPICSDataBlockOffset:=92);

        //********************************************
        // Device name: Spk-000CDL:Cryo-PID-91
        // Device type: C3S_PID
        //********************************************

      "DEV_Spk-000CDL:Cryo-PID-91_iDB" (EPICSToPLCLength:=26,
      EPICSToPLCDataBlockOffset:=86,
      PLCToEPICSLength:=90,
      PLCToEPICSDataBlockOffset:=117);

        //********************************************
        // Device name: Spk-000CDL:Cryo-PID-92
        // Device type: C3S_PID
        //********************************************

      "DEV_Spk-000CDL:Cryo-PID-92_iDB" (EPICSToPLCLength:=26,
      EPICSToPLCDataBlockOffset:=112,
      PLCToEPICSLength:=90,
      PLCToEPICSDataBlockOffset:=207);

        //********************************************
        // Device name: Spk-000CDL:Cryo-PID-93
        // Device type: C3S_PID
        //********************************************

      "DEV_Spk-000CDL:Cryo-PID-93_iDB" (EPICSToPLCLength:=26,
      EPICSToPLCDataBlockOffset:=138,
      PLCToEPICSLength:=90,
      PLCToEPICSDataBlockOffset:=297);

        //********************************************
        // Device name: Spk-000CDL:Cryo-PID-94
        // Device type: C3S_PID
        //********************************************

      "DEV_Spk-000CDL:Cryo-PID-94_iDB" (EPICSToPLCLength:=26,
      EPICSToPLCDataBlockOffset:=164,
      PLCToEPICSLength:=90,
      PLCToEPICSDataBlockOffset:=387);

        //********************************************
        // Device name: Spk-000CDL:Cryo-CV-91
        // Device type: ICS_CV_PB_SIPART
        //********************************************

      "DEV_Spk-000CDL:Cryo-CV-91_iDB" (EPICSToPLCLength:=23,
      EPICSToPLCDataBlockOffset:=190,
      PLCToEPICSLength:=75,
      PLCToEPICSDataBlockOffset:=477);

        //********************************************
        // Device name: Spk-000CDL:Cryo-CV-92
        // Device type: ICS_CV_PB_SIPART
        //********************************************

      "DEV_Spk-000CDL:Cryo-CV-92_iDB" (EPICSToPLCLength:=23,
      EPICSToPLCDataBlockOffset:=213,
      PLCToEPICSLength:=75,
      PLCToEPICSDataBlockOffset:=552);

        //********************************************
        // Device name: Spk-000CDL:Cryo-CV-93
        // Device type: ICS_CV_PB_SIPART
        //********************************************

      "DEV_Spk-000CDL:Cryo-CV-93_iDB" (EPICSToPLCLength:=23,
      EPICSToPLCDataBlockOffset:=236,
      PLCToEPICSLength:=75,
      PLCToEPICSDataBlockOffset:=627);

        //********************************************
        // Device name: Spk-000CDL:Cryo-CV-94
        // Device type: ICS_CV_PB_SIPART
        //********************************************

      "DEV_Spk-000CDL:Cryo-CV-94_iDB" (EPICSToPLCLength:=23,
      EPICSToPLCDataBlockOffset:=259,
      PLCToEPICSLength:=75,
      PLCToEPICSDataBlockOffset:=702);

        //********************************************
        // Device name: Spk-000CDL:Cryo-EH-91
        // Device type: ICS_EH
        //********************************************

      "DEV_Spk-000CDL:Cryo-EH-91_iDB" (EPICSToPLCLength:=19,
      EPICSToPLCDataBlockOffset:=282,
      PLCToEPICSLength:=45,
      PLCToEPICSDataBlockOffset:=777);

        //********************************************
        // Device name: Spk-000CDL:Cryo-EH-92
        // Device type: ICS_EH
        //********************************************

      "DEV_Spk-000CDL:Cryo-EH-92_iDB" (EPICSToPLCLength:=19,
      EPICSToPLCDataBlockOffset:=301,
      PLCToEPICSLength:=45,
      PLCToEPICSDataBlockOffset:=822);

        //********************************************
        // Device name: Spk-000CDL:Cryo-EH-93
        // Device type: ICS_EH
        //********************************************

      "DEV_Spk-000CDL:Cryo-EH-93_iDB" (EPICSToPLCLength:=19,
      EPICSToPLCDataBlockOffset:=320,
      PLCToEPICSLength:=45,
      PLCToEPICSDataBlockOffset:=867);

        //********************************************
        // Device name: Spk-000CDL:Cryo-EH-94
        // Device type: ICS_EH
        //********************************************

      "DEV_Spk-000CDL:Cryo-EH-94_iDB" (EPICSToPLCLength:=19,
      EPICSToPLCDataBlockOffset:=339,
      PLCToEPICSLength:=45,
      PLCToEPICSDataBlockOffset:=912);

        //********************************************
        // Device name: Spk-000CDL:Cryo-EH-95
        // Device type: ICS_EH
        //********************************************

      "DEV_Spk-000CDL:Cryo-EH-95_iDB" (EPICSToPLCLength:=19,
      EPICSToPLCDataBlockOffset:=358,
      PLCToEPICSLength:=45,
      PLCToEPICSDataBlockOffset:=957);

        //********************************************
        // Device name: Spk-000CDL:Cryo-EH-96
        // Device type: ICS_EH
        //********************************************

      "DEV_Spk-000CDL:Cryo-EH-96_iDB" (EPICSToPLCLength:=19,
      EPICSToPLCDataBlockOffset:=377,
      PLCToEPICSLength:=45,
      PLCToEPICSDataBlockOffset:=1002);

        //********************************************
        // Device name: Spk-000CDL:Cryo-HV-70
        // Device type: ICS_HV
        //********************************************

      "DEV_Spk-000CDL:Cryo-HV-70_iDB" (EPICSToPLCLength:=5,
      EPICSToPLCDataBlockOffset:=396,
      PLCToEPICSLength:=8,
      PLCToEPICSDataBlockOffset:=1047);

        //********************************************
        // Device name: Spk-000CDL:Cryo-HV-73
        // Device type: ICS_HV
        //********************************************

      "DEV_Spk-000CDL:Cryo-HV-73_iDB" (EPICSToPLCLength:=5,
      EPICSToPLCDataBlockOffset:=401,
      PLCToEPICSLength:=8,
      PLCToEPICSDataBlockOffset:=1055);

        //********************************************
        // Device name: Spk-000CDL:Cryo-TT-91
        // Device type: ICS_LAKESHORE_TT
        //********************************************

      "DEV_Spk-000CDL:Cryo-TT-91_iDB" (EPICSToPLCLength:=15,
      EPICSToPLCDataBlockOffset:=406,
      PLCToEPICSLength:=25,
      PLCToEPICSDataBlockOffset:=1063);

        //********************************************
        // Device name: Spk-000CDL:Cryo-TT-92
        // Device type: ICS_LAKESHORE_TT
        //********************************************

      "DEV_Spk-000CDL:Cryo-TT-92_iDB" (EPICSToPLCLength:=15,
      EPICSToPLCDataBlockOffset:=421,
      PLCToEPICSLength:=25,
      PLCToEPICSDataBlockOffset:=1088);

        //********************************************
        // Device name: Spk-000CDL:Cryo-TT-93
        // Device type: ICS_LAKESHORE_TT
        //********************************************

      "DEV_Spk-000CDL:Cryo-TT-93_iDB" (EPICSToPLCLength:=15,
      EPICSToPLCDataBlockOffset:=436,
      PLCToEPICSLength:=25,
      PLCToEPICSDataBlockOffset:=1113);

        //********************************************
        // Device name: Spk-000CDL:Cryo-TT-94
        // Device type: ICS_LAKESHORE_TT
        //********************************************

      "DEV_Spk-000CDL:Cryo-TT-94_iDB" (EPICSToPLCLength:=15,
      EPICSToPLCDataBlockOffset:=451,
      PLCToEPICSLength:=25,
      PLCToEPICSDataBlockOffset:=1138);

        //********************************************
        // Device name: Spk-000CDL:Cryo-TT-95
        // Device type: ICS_LAKESHORE_TT
        //********************************************

      "DEV_Spk-000CDL:Cryo-TT-95_iDB" (EPICSToPLCLength:=15,
      EPICSToPLCDataBlockOffset:=466,
      PLCToEPICSLength:=25,
      PLCToEPICSDataBlockOffset:=1163);

        //********************************************
        // Device name: Spk-000CDL:Cryo-TT-96
        // Device type: ICS_LAKESHORE_TT
        //********************************************

      "DEV_Spk-000CDL:Cryo-TT-96_iDB" (EPICSToPLCLength:=15,
      EPICSToPLCDataBlockOffset:=481,
      PLCToEPICSLength:=25,
      PLCToEPICSDataBlockOffset:=1188);

        //********************************************
        // Device name: Spk-000CDL:Cryo-TT-97
        // Device type: ICS_LAKESHORE_TT
        //********************************************

      "DEV_Spk-000CDL:Cryo-TT-97_iDB" (EPICSToPLCLength:=15,
      EPICSToPLCDataBlockOffset:=496,
      PLCToEPICSLength:=25,
      PLCToEPICSDataBlockOffset:=1213);

        //********************************************
        // Device name: Spk-000CDL:Cryo-TT-98
        // Device type: ICS_LAKESHORE_TT
        //********************************************

      "DEV_Spk-000CDL:Cryo-TT-98_iDB" (EPICSToPLCLength:=15,
      EPICSToPLCDataBlockOffset:=511,
      PLCToEPICSLength:=25,
      PLCToEPICSDataBlockOffset:=1238);

        //********************************************
        // Device name: Spk-000CDL:Cryo-LT-91
        // Device type: ICS_LT
        //********************************************

      "DEV_Spk-000CDL:Cryo-LT-91_iDB" (EPICSToPLCLength:=23,
      EPICSToPLCDataBlockOffset:=526,
      PLCToEPICSLength:=32,
      PLCToEPICSDataBlockOffset:=1263);

        //********************************************
        // Device name: Spk-000CDL:Cryo-LT-92
        // Device type: ICS_LT
        //********************************************

      "DEV_Spk-000CDL:Cryo-LT-92_iDB" (EPICSToPLCLength:=23,
      EPICSToPLCDataBlockOffset:=549,
      PLCToEPICSLength:=32,
      PLCToEPICSDataBlockOffset:=1295);

        //********************************************
        // Device name: Spk-000CDL:Cryo-PT-91
        // Device type: ICS_PT_mbar
        //********************************************

